  MoveL 8252 to (508.91, 501.9, 16.3) mm, rotated rx 0 ry 90 rz 0 deg; joints [-12.009, -27.828, 110.474, -16.064, -82.068, 51.258]
  Set speed (15.0 mm/s)
  Call Extruder(0.081)
  MoveL 8253 to (508.91, 504.67, 16.3) mm, rotated rx 0 ry 90 rz 0 deg; joints [-12.259, -27.816, 110.402, -16.319, -82.019, 51.306]
  Call Extruder(0.035)
  MoveL 8254 to (507.71, 504.67, 16.3) mm, rotated rx 0 ry 90 rz 0 deg; joints [-12.282, -27.84, 110.547, -16.337, -82.135, 51.275]
  Call Extruder(0.081)
  MoveL 8255 to (507.71, 501.9, 16.3) mm, rotated rx 0 ry 90 rz 0 deg; joints [-12.032, -27.852, 110.619, -16.082, -82.184, 51.227]
  Call Extruder(0.035)
  MoveL 8256 to (508.91, 501.9, 16.3) mm, rotated rx 0 ry 90 rz 0 deg; joints [-12.009, -27.828, 110.474, -16.064, -82.068, 51.258]
  Set speed (120.0 mm/s)
  MoveL 8257 to (508.59, 502.65, 16.3) mm, rotated rx 0 ry 90 rz 0 deg; joints [-12.083, -27.831, 110.493, -16.138, -82.085, 51.263]
  Set speed (15.0 mm/s)
  Call Extruder(0.018)
  MoveL 8258 to (508.15, 502.21, 16.3) mm, rotated rx 0 ry 90 rz 0 deg; joints [-12.052, -27.842, 110.557, -16.105, -82.136, 51.244]
  Set speed (120.0 mm/s)
  MoveL 8259 to (508.02, 503.08, 16.3) mm, rotated rx 0 ry 90 rz 0 deg; joints [-12.132, -27.841, 110.55, -16.186, -82.133, 51.255]
  Set speed (15.0 mm/s)
  Call Extruder(0.023)
  MoveL 8260 to (508.59, 503.64, 16.3) mm, rotated rx 0 ry 90 rz 0 deg; joints [-12.172, -27.827, 110.467, -16.229, -82.068, 51.28]
  Set speed (120.0 mm/s)
  MoveL 8261 to (508.02, 504.07, 16.3) mm, rotated rx 0 ry 90 rz 0 deg; joints [-12.222, -27.836, 110.525, -16.277, -82.116, 51.272]
  Set speed (15.0 mm/s)
  Call Extruder(0.012)
  MoveL 8262 to (508.32, 504.36, 16.3) mm, rotated rx 0 ry 90 rz 0 deg; joints [-12.242, -27.829, 110.482, -16.299, -82.082, 51.285]
  Set speed (120.0 mm/s)
  MoveL 8263 to (490.68, 490.68, 16.3) mm, rotated rx 0 ry 90 rz 0 deg; joints [-11.324, -28.211, 112.929, -15.306, -84.042, 50.621]
  Set speed (1000.0 mm/s)
  MoveL 8264 to (490.68, 490.68, 16.4) mm, rotated rx 0 ry 90 rz 0 deg; joints [-11.324, -28.222, 112.934, -15.306, -84.036, 50.622]
  Set speed (30.0 mm/s)
  Call Extruder(0.767)
  MoveL 8265 to (509.32, 509.32, 16.4) mm, rotated rx 0 ry 90 rz 0 deg; joints [-12.669, -27.797, 110.234, -16.738, -81.892, 51.4]
  MoveL 8266 to (509.44, 509.44, 16.4) mm, rotated rx 0 ry 90 rz 0 deg; joints [-12.677, -27.794, 110.216, -16.747, -81.878, 51.406]
  Set speed (120.0 mm/s)
  MoveL 8267 to (507.79, 502.11, 16.4) mm, rotated rx 0 ry 90 rz 0 deg; joints [-12.049, -27.86, 110.609, -16.101, -82.168, 51.234]
  Set speed (30.0 mm/s)
  Call Extruder(0.297)
  MoveL 8268 to (500.58, 509.32, 16.4) mm, rotated rx 0 ry 90 rz 0 deg; joints [-12.847, -27.971, 111.282, -16.884, -82.735, 51.167]
  Set speed (120.0 mm/s)
  MoveL 8269 to (499.42, 509.32, 16.4) mm, rotated rx 0 ry 90 rz 0 deg; joints [-12.872, -27.993, 111.421, -16.904, -82.847, 51.135]
  Set speed (30.0 mm/s)
  Call Extruder(0.360)
  MoveL 8270 to (490.68, 500.58, 16.4) mm, rotated rx 0 ry 90 rz 0 deg; joints [-12.247, -28.186, 112.689, -16.24, -83.859, 50.763]
  Set speed (120.0 mm/s)
  MoveL 8271 to (490.68, 499.42, 16.4) mm, rotated rx 0 ry 90 rz 0 deg; joints [-12.139, -28.191, 112.719, -16.13, -83.88, 50.746]
  Set speed (30.0 mm/s)
  MoveL 8272 to (499.42, 490.68, 16.4) mm, rotated rx 0 ry 90 rz 0 deg; joints [-11.163, -28.067, 111.894, -15.17, -83.178, 50.841]
  Set speed (120.0 mm/s)
  MoveL 8273 to (500.58, 490.68, 16.4) mm, rotated rx 0 ry 90 rz 0 deg; joints [-11.142, -28.046, 111.756, -15.152, -83.065, 50.869]
  Set speed (30.0 mm/s)
  Call Extruder(0.055)
  MoveL 8274 to (501.92, 492.02, 16.4) mm, rotated rx 0 ry 90 rz 0 deg; joints [-11.24, -28.016, 111.564, -15.257, -82.912, 50.923]
  Set speed (120.0 mm/s)
  MoveL 8275 to (502.08, 492.18, 16.4) mm, rotated rx 0 ry 90 rz 0 deg; joints [-11.252, -28.012, 111.54, -15.27, -82.893, 50.929]
  Set speed (30.0 mm/s)
  Call Extruder(0.298)
  MoveL 8276 to (509.32, 499.42, 16.4) mm, rotated rx 0 ry 90 rz 0 deg; joints [-11.777, -27.841, 110.493, -15.83, -82.065, 51.227]
  Set speed (120.0 mm/s)
  MoveL 8277 to (509.32, 500.58, 16.4) mm, rotated rx 0 ry 90 rz 0 deg; joints [-11.882, -27.836, 110.463, -15.936, -82.046, 51.247]
  Set speed (30.0 mm/s)
  Call Extruder(0.060)
  MoveL 8278 to (507.86, 502.04, 16.4) mm, rotated rx 0 ry 90 rz 0 deg; joints [-12.041, -27.859, 110.602, -16.093, -82.162, 51.235]
  MoveL 8279 to (507.74, 502.16, 16.4) mm, rotated rx 0 ry 90 rz 0 deg; joints [-12.055, -27.861, 110.613, -16.106, -82.172, 51.234]
  Set speed (120.0 mm/s)
  MoveL 8280 to (509.32, 490.68, 16.4) mm, rotated rx 0 ry 90 rz 0 deg; joints [-10.985, -27.876, 110.705, -15.024, -82.209, 51.083]
  Set speed (30.0 mm/s)
  Call Extruder(0.767)
  MoveL 8281 to (490.68, 509.32, 16.4) mm, rotated rx 0 ry 90 rz 0 deg; joints [-13.056, -28.152, 112.457, -17.059, -83.692, 50.896]
  MoveL 8282 to (490.56, 509.44, 16.4) mm, rotated rx 0 ry 90 rz 0 deg; joints [-13.07, -28.154, 112.469, -17.073, -83.701, 50.895]
  Set speed (120.0 mm/s)
  MoveL 8283 to (490.4, 509.6, 16.4) mm, rotated rx 0 ry 90 rz 0 deg; joints [-13.088, -28.156, 112.483, -17.091, -83.713, 50.893]
  Set speed (15.0 mm/s)
  Call Extruder(0.559)
  MoveL 8284 to (490.4, 490.4, 16.4) mm, rotated rx 0 ry 90 rz 0 deg; joints [-11.303, -28.227, 112.973, -15.284, -84.068, 50.611]
  MoveL 8285 to (509.6, 490.4, 16.4) mm, rotated rx 0 ry 90 rz 0 deg; joints [-10.955, -27.872, 110.678, -14.995, -82.186, 51.085]
  MoveL 8286 to (509.6, 509.6, 16.4) mm, rotated rx 0 ry 90 rz 0 deg; joints [-12.688, -27.79, 110.193, -16.759, -81.86, 51.413]
  MoveL 8287 to (490.4, 509.6, 16.4) mm, rotated rx 0 ry 90 rz 0 deg; joints [-13.088, -28.156, 112.483, -17.091, -83.713, 50.893]
  Set speed (120.0 mm/s)
  MoveL 8288 to (490.4, 509.2, 16.4) mm, rotated rx 0 ry 90 rz 0 deg; joints [-13.051, -28.158, 112.494, -17.053, -83.721, 50.887]
  Set speed (1000.0 mm/s)
  MoveL 8289 to (490.5, 509.2, 16.4) mm, rotated rx 0 ry 90 rz 0 deg; joints [-13.049, -28.156, 112.482, -17.052, -83.711, 50.89]
  Set speed (1000.0 mm/s)
  MoveL 8290 to (494.92, 492.25, 16.4) mm, rotated rx 0 ry 90 rz 0 deg; joints [-11.391, -28.143, 112.393, -15.387, -83.593, 50.751]
  Set speed (15.0 mm/s)
  Call Extruder(0.034)
  MoveL 8291 to (494.92, 491.09, 16.4) mm, rotated rx 0 ry 90 rz 0 deg; joints [-11.283, -28.147, 112.421, -15.278, -83.613, 50.735]
  Call Extruder(0.076)
  MoveL 8292 to (497.51, 491.09, 16.4) mm, rotated rx 0 ry 90 rz 0 deg; joints [-11.235, -28.101, 112.112, -15.237, -83.358, 50.799]
  Call Extruder(0.034)
  MoveL 8293 to (497.51, 492.26, 16.4) mm, rotated rx 0 ry 90 rz 0 deg; joints [-11.344, -28.096, 112.084, -15.347, -83.339, 50.817]
  Call Extruder(0.074)
  MoveL 8294 to (494.97, 492.26, 16.4) mm, rotated rx 0 ry 90 rz 0 deg; joints [-11.391, -28.142, 112.387, -15.387, -83.587, 50.753]
  Call Extruder(0.000)
  MoveL 8295 to (494.97, 492.25, 16.4) mm, rotated rx 0 ry 90 rz 0 deg; joints [-11.39, -28.142, 112.387, -15.386, -83.587, 50.753]
  Call Extruder(0.002)
  MoveL 8296 to (494.92, 492.25, 16.4) mm, rotated rx 0 ry 90 rz 0 deg; joints [-11.391, -28.143, 112.393, -15.387, -83.593, 50.751]
  Set speed (120.0 mm/s)
  MoveL 8297 to (495.23, 491.75, 16.4) mm, rotated rx 0 ry 90 rz 0 deg; joints [-11.339, -28.139, 112.368, -15.335, -83.571, 50.752]
  Set speed (15.0 mm/s)
  Call Extruder(0.014)
  MoveL 8298 to (495.58, 491.4, 16.4) mm, rotated rx 0 ry 90 rz 0 deg; joints [-11.3, -28.134, 112.335, -15.297, -83.543, 50.756]
  Set speed (120.0 mm/s)
  MoveL 8299 to (496.02, 491.95, 16.4) mm, rotated rx 0 ry 90 rz 0 deg; joints [-11.342, -28.124, 112.269, -15.341, -83.49, 50.775]
  Set speed (15.0 mm/s)
  Call Extruder(0.022)
  MoveL 8300 to (496.57, 491.4, 16.4) mm, rotated rx 0 ry 90 rz 0 deg; joints [-11.282, -28.117, 112.218, -15.281, -83.446, 50.78]
  Set speed (120.0 mm/s)
  MoveL 8301 to (497.01, 491.95, 16.4) mm, rotated rx 0 ry 90 rz 0 deg; joints [-11.324, -28.107, 112.151, -15.325, -83.393, 50.799]
  Set speed (15.0 mm/s)
  Call Extruder(0.008)
  MoveL 8302 to (497.2, 491.76, 16.4) mm, rotated rx 0 ry 90 rz 0 deg; joints [-11.303, -28.104, 112.134, -15.305, -83.378, 50.801]
  Set speed (120.0 mm/s)
  MoveL 8303 to (501.84, 492.26, 16.4) mm, rotated rx 0 ry 90 rz 0 deg; joints [-11.264, -28.016, 111.568, -15.281, -82.915, 50.924]
  Set speed (15.0 mm/s)
  Call Extruder(0.034)
  MoveL 8304 to (501.84, 491.09, 16.4) mm, rotated rx 0 ry 90 rz 0 deg; joints [-11.157, -28.021, 111.595, -15.172, -82.935, 50.906]
  Call Extruder(0.076)
  MoveL 8305 to (504.46, 491.09, 16.4) mm, rotated rx 0 ry 90 rz 0 deg; joints [-11.109, -27.971, 111.281, -15.133, -82.678, 50.971]
  Call Extruder(0.034)
  MoveL 8306 to (504.46, 492.27, 16.4) mm, rotated rx 0 ry 90 rz 0 deg; joints [-11.217, -27.966, 111.253, -15.242, -82.659, 50.989]
  Call Extruder(0.016)
  MoveL 8307 to (503.92, 492.26, 16.4) mm, rotated rx 0 ry 90 rz 0 deg; joints [-11.226, -27.976, 111.317, -15.25, -82.711, 50.976]
  Call Extruder(0.061)
  MoveL 8308 to (501.84, 492.26, 16.4) mm, rotated rx 0 ry 90 rz 0 deg; joints [-11.264, -28.016, 111.568, -15.281, -82.915, 50.924]
  Set speed (120.0 mm/s)
  MoveL 8309 to (502.15, 491.76, 16.4) mm, rotated rx 0 ry 90 rz 0 deg; joints [-11.212, -28.012, 111.542, -15.229, -82.893, 50.924]
  Set speed (15.0 mm/s)
  Call Extruder(0.015)
  MoveL 8310 to (502.5, 491.4, 16.4) mm, rotated rx 0 ry 90 rz 0 deg; joints [-11.173, -28.007, 111.508, -15.191, -82.864, 50.928]
  Set speed (120.0 mm/s)
  MoveL 8311 to (502.95, 491.95, 16.4) mm, rotated rx 0 ry 90 rz 0 deg; joints [-11.215, -27.996, 111.441, -15.235, -82.811, 50.947]
  Set speed (15.0 mm/s)
  Call Extruder(0.022)
  MoveL 8312 to (503.49, 491.4, 16.4) mm, rotated rx 0 ry 90 rz 0 deg; joints [-11.155, -27.988, 111.389, -15.176, -82.767, 50.952]
  Set speed (120.0 mm/s)
  MoveL 8313 to (503.94, 491.95, 16.4) mm, rotated rx 0 ry 90 rz 0 deg; joints [-11.197, -27.977, 111.323, -15.22, -82.714, 50.972]
  Set speed (15.0 mm/s)
  Call Extruder(0.008)
  MoveL 8314 to (504.14, 491.75, 16.4) mm, rotated rx 0 ry 90 rz 0 deg; joints [-11.175, -27.974, 111.303, -15.198, -82.698, 50.973]
  Set speed (120.0 mm/s)
  MoveL 8315 to (507.71, 494.38, 16.4) mm, rotated rx 0 ry 90 rz 0 deg; joints [-11.351, -27.894, 110.81, -15.39, -82.306, 51.104]
  Set speed (15.0 mm/s)
  Call Extruder(0.035)
  MoveL 8316 to (508.91, 494.38, 16.4) mm, rotated rx 0 ry 90 rz 0 deg; joints [-11.328, -27.87, 110.667, -15.371, -82.189, 51.133]
  Call Extruder(0.079)
  MoveL 8317 to (508.91, 497.08, 16.4) mm, rotated rx 0 ry 90 rz 0 deg; joints [-11.573, -27.859, 110.601, -15.62, -82.145, 51.178]
  Call Extruder(0.035)
  MoveL 8318 to (507.71, 497.08, 16.4) mm, rotated rx 0 ry 90 rz 0 deg; joints [-11.595, -27.883, 110.745, -15.638, -82.261, 51.148]
  Call Extruder(0.051)
  MoveL 8319 to (507.71, 495.33, 16.4) mm, rotated rx 0 ry 90 rz 0 deg; joints [-11.437, -27.89, 110.788, -15.477, -82.29, 51.119]
  Call Extruder(0.028)
  MoveL 8320 to (507.71, 494.38, 16.4) mm, rotated rx 0 ry 90 rz 0 deg; joints [-11.351, -27.894, 110.81, -15.39, -82.306, 51.104]
  Set speed (120.0 mm/s)
  MoveL 8321 to (508.59, 495.21, 16.4) mm, rotated rx 0 ry 90 rz 0 deg; joints [-11.41, -27.873, 110.684, -15.453, -82.206, 51.139]
  Set speed (15.0 mm/s)
  Call Extruder(0.023)
  MoveL 8322 to (508.03, 495.78, 16.4) mm, rotated rx 0 ry 90 rz 0 deg; joints [-11.472, -27.882, 110.739, -15.514, -82.252, 51.134]
  Set speed (120.0 mm/s)
  MoveL 8323 to (508.59, 496.2, 16.4) mm, rotated rx 0 ry 90 rz 0 deg; joints [-11.5, -27.869, 110.66, -15.545, -82.19, 51.155]
  Set speed (15.0 mm/s)
  Call Extruder(0.023)
  MoveL 8324 to (508.04, 496.76, 16.4) mm, rotated rx 0 ry 90 rz 0 deg; joints [-11.56, -27.878, 110.714, -15.604, -82.235, 51.151]
  Set speed (120.0 mm/s)
  MoveL 8325 to (507.71, 501.95, 16.4) mm, rotated rx 0 ry 90 rz 0 deg; joints [-12.037, -27.862, 110.622, -16.088, -82.178, 51.23]
  Set speed (15.0 mm/s)
  Call Extruder(0.035)
  MoveL 8326 to (508.91, 501.96, 16.4) mm, rotated rx 0 ry 90 rz 0 deg; joints [-12.014, -27.838, 110.478, -16.069, -82.062, 51.26]
  Call Extruder(0.079)
  MoveL 8327 to (508.91, 504.67, 16.4) mm, rotated rx 0 ry 90 rz 0 deg; joints [-12.259, -27.826, 110.407, -16.319, -82.014, 51.307]
  Call Extruder(0.035)
  MoveL 8328 to (507.71, 504.67, 16.4) mm, rotated rx 0 ry 90 rz 0 deg; joints [-12.282, -27.851, 110.552, -16.338, -82.13, 51.276]
  Call Extruder(0.079)
  MoveL 8329 to (507.71, 501.95, 16.4) mm, rotated rx 0 ry 90 rz 0 deg; joints [-12.037, -27.862, 110.622, -16.088, -82.178, 51.23]
  Set speed (120.0 mm/s)
  MoveL 8330 to (508.03, 502.71, 16.4) mm, rotated rx 0 ry 90 rz 0 deg; joints [-12.099, -27.853, 110.565, -16.153, -82.134, 51.251]
  Set speed (15.0 mm/s)
  Call Extruder(0.018)
  MoveL 8331 to (508.47, 502.27, 16.4) mm, rotated rx 0 ry 90 rz 0 deg; joints [-12.051, -27.846, 110.523, -16.105, -82.099, 51.254]
  Set speed (120.0 mm/s)
  MoveL 8332 to (508.59, 503.13, 16.4) mm, rotated rx 0 ry 90 rz 0 deg; joints [-12.126, -27.839, 110.485, -16.182, -82.072, 51.273]
  Set speed (15.0 mm/s)
  Call Extruder(0.023)
  MoveL 8333 to (508.02, 503.7, 16.4) mm, rotated rx 0 ry 90 rz 0 deg; joints [-12.189, -27.848, 110.539, -16.244, -82.117, 51.268]
  Set speed (120.0 mm/s)
  MoveL 8334 to (508.59, 504.12, 16.4) mm, rotated rx 0 ry 90 rz 0 deg; joints [-12.216, -27.835, 110.46, -16.273, -82.054, 51.29]
  Set speed (15.0 mm/s)
  Call Extruder(0.010)
  MoveL 8335 to (508.36, 504.36, 16.4) mm, rotated rx 0 ry 90 rz 0 deg; joints [-12.241, -27.839, 110.482, -16.299, -82.073, 51.288]
  Set speed (120.0 mm/s)
  MoveL 8336 to (490.68, 490.68, 16.4) mm, rotated rx 0 ry 90 rz 0 deg; joints [-11.324, -28.222, 112.934, -15.306, -84.036, 50.622]
  Set speed (1000.0 mm/s)
  MoveL 8337 to (490.68, 490.68, 16.5) mm, rotated rx 0 ry 90 rz 0 deg; joints [-11.324, -28.232, 112.939, -15.306, -84.031, 50.624]
  Set speed (30.0 mm/s)
  Call Extruder(0.767)
  MoveL 8338 to (509.32, 509.32, 16.5) mm, rotated rx 0 ry 90 rz 0 deg; joints [-12.669, -27.807, 110.239, -16.738, -81.887, 51.402]
  MoveL 8339 to (509.44, 509.44, 16.5) mm, rotated rx 0 ry 90 rz 0 deg; joints [-12.677, -27.804, 110.221, -16.747, -81.873, 51.407]
  Set speed (120.0 mm/s)
  MoveL 8340 to (507.79, 502.11, 16.5) mm, rotated rx 0 ry 90 rz 0 deg; joints [-12.049, -27.871, 110.614, -16.101, -82.162, 51.236]
  Set speed (30.0 mm/s)
  Call Extruder(0.297)
  MoveL 8341 to (500.58, 509.32, 16.5) mm, rotated rx 0 ry 90 rz 0 deg; joints [-12.847, -27.981, 111.287, -16.884, -82.73, 51.168]
  Set speed (120.0 mm/s)
  MoveL 8342 to (499.42, 509.32, 16.5) mm, rotated rx 0 ry 90 rz 0 deg; joints [-12.872, -28.003, 111.426, -16.904, -82.842, 51.137]
  Set speed (30.0 mm/s)
  Call Extruder(0.360)
  MoveL 8343 to (490.68, 500.58, 16.5) mm, rotated rx 0 ry 90 rz 0 deg; joints [-12.247, -28.197, 112.694, -16.24, -83.853, 50.765]
  Set speed (120.0 mm/s)
  MoveL 8344 to (490.68, 499.42, 16.5) mm, rotated rx 0 ry 90 rz 0 deg; joints [-12.139, -28.201, 112.724, -16.131, -83.875, 50.748]
  Set speed (30.0 mm/s)
  MoveL 8345 to (499.42, 490.68, 16.5) mm, rotated rx 0 ry 90 rz 0 deg; joints [-11.163, -28.078, 111.899, -15.17, -83.173, 50.842]
  Set speed (120.0 mm/s)
  MoveL 8346 to (500.58, 490.68, 16.5) mm, rotated rx 0 ry 90 rz 0 deg; joints [-11.141, -28.056, 111.761, -15.152, -83.059, 50.871]
  Set speed (30.0 mm/s)
  Call Extruder(0.058)
  MoveL 8347 to (501.98, 492.08, 16.5) mm, rotated rx 0 ry 90 rz 0 deg; joints [-11.245, -28.025, 111.56, -15.262, -82.899, 50.927]
  Set speed (120.0 mm/s)
  MoveL 8348 to (502.08, 492.18, 16.5) mm, rotated rx 0 ry 90 rz 0 deg; joints [-11.252, -28.022, 111.545, -15.27, -82.887, 50.931]
  Set speed (30.0 mm/s)
  Call Extruder(0.298)
  MoveL 8349 to (509.32, 499.42, 16.5) mm, rotated rx 0 ry 90 rz 0 deg; joints [-11.777, -27.851, 110.498, -15.83, -82.06, 51.229]
  Set speed (120.0 mm/s)
  MoveL 8350 to (509.32, 500.58, 16.5) mm, rotated rx 0 ry 90 rz 0 deg; joints [-11.882, -27.846, 110.469, -15.937, -82.04, 51.249]
  Set speed (30.0 mm/s)
  Call Extruder(0.062)
  MoveL 8351 to (507.81, 502.09, 16.5) mm, rotated rx 0 ry 90 rz 0 deg; joints [-12.047, -27.87, 110.612, -16.099, -82.161, 51.236]
  MoveL 8352 to (507.69, 502.21, 16.5) mm, rotated rx 0 ry 90 rz 0 deg; joints [-12.061, -27.872, 110.624, -16.112, -82.171, 51.235]
  Set speed (120.0 mm/s)
  MoveL 8353 to (509.32, 490.68, 16.5) mm, rotated rx 0 ry 90 rz 0 deg; joints [-10.985, -27.887, 110.71, -15.025, -82.204, 51.084]
  Set speed (30.0 mm/s)
  Call Extruder(0.767)
  MoveL 8354 to (490.68, 509.32, 16.5) mm, rotated rx 0 ry 90 rz 0 deg; joints [-13.056, -28.163, 112.463, -17.06, -83.686, 50.898]
  MoveL 8355 to (490.56, 509.44, 16.5) mm, rotated rx 0 ry 90 rz 0 deg; joints [-13.07, -28.165, 112.474, -17.073, -83.696, 50.897]
  Set speed (120.0 mm/s)
  MoveL 8356 to (490.4, 509.6, 16.5) mm, rotated rx 0 ry 90 rz 0 deg; joints [-13.088, -28.167, 112.488, -17.091, -83.708, 50.895]
  Set speed (15.0 mm/s)
  Call Extruder(0.559)
  MoveL 8357 to (490.4, 490.4, 16.5) mm, rotated rx 0 ry 90 rz 0 deg; joints [-11.303, -28.238, 112.978, -15.284, -84.063, 50.613]
  MoveL 8358 to (509.6, 490.4, 16.5) mm, rotated rx 0 ry 90 rz 0 deg; joints [-10.955, -27.882, 110.683, -14.995, -82.181, 51.086]
  MoveL 8359 to (509.6, 509.6, 16.5) mm, rotated rx 0 ry 90 rz 0 deg; joints [-12.688, -27.8, 110.198, -16.759, -81.855, 51.414]
  MoveL 8360 to (490.4, 509.6, 16.5) mm, rotated rx 0 ry 90 rz 0 deg; joints [-13.088, -28.167, 112.488, -17.091, -83.708, 50.895]
  Set speed (120.0 mm/s)
  MoveL 8361 to (490.4, 509.2, 16.5) mm, rotated rx 0 ry 90 rz 0 deg; joints [-13.051, -28.168, 112.499, -17.054, -83.716, 50.888]
  Set speed (1000.0 mm/s)
  MoveL 8362 to (490.5, 509.2, 16.5) mm, rotated rx 0 ry 90 rz 0 deg; joints [-13.049, -28.167, 112.487, -17.052, -83.706, 50.891]
  Set speed (1000.0 mm/s)
  MoveL 8363 to (494.92, 492.25, 16.5) mm, rotated rx 0 ry 90 rz 0 deg; joints [-11.391, -28.154, 112.399, -15.387, -83.588, 50.753]
  Set speed (15.0 mm/s)
  Call Extruder(0.034)
  MoveL 8364 to (494.92, 491.09, 16.5) mm, rotated rx 0 ry 90 rz 0 deg; joints [-11.283, -28.158, 112.426, -15.278, -83.608, 50.736]
  Call Extruder(0.074)
  MoveL 8365 to (497.46, 491.09, 16.5) mm, rotated rx 0 ry 90 rz 0 deg; joints [-11.236, -28.112, 112.124, -15.238, -83.358, 50.799]
  Call Extruder(0.034)
  MoveL 8366 to (497.45, 492.26, 16.5) mm, rotated rx 0 ry 90 rz 0 deg; joints [-11.345, -28.108, 112.096, -15.348, -83.339, 50.817]
  Call Extruder(0.072)
  MoveL 8367 to (494.97, 492.26, 16.5) mm, rotated rx 0 ry 90 rz 0 deg; joints [-11.391, -28.152, 112.392, -15.387, -83.582, 50.754]
  Call Extruder(0.000)
  MoveL 8368 to (494.97, 492.25, 16.5) mm, rotated rx 0 ry 90 rz 0 deg; joints [-11.39, -28.153, 112.392, -15.386, -83.582, 50.754]
  Call Extruder(0.002)
  MoveL 8369 to (494.92, 492.25, 16.5) mm, rotated rx 0 ry 90 rz 0 deg; joints [-11.391, -28.154, 112.399, -15.387, -83.588, 50.753]
  Set speed (120.0 mm/s)
  MoveL 8370 to (495.37, 491.41, 16.5) mm, rotated rx 0 ry 90 rz 0 deg; joints [-11.304, -28.149, 112.365, -15.3, -83.558, 50.752]
  Set speed (15.0 mm/s)
  Call Extruder(0.022)
  MoveL 8371 to (495.91, 491.95, 16.5) mm, rotated rx 0 ry 90 rz 0 deg; joints [-11.344, -28.137, 112.288, -15.343, -83.496, 50.773]
  Set speed (120.0 mm/s)
  MoveL 8372 to (496.36, 491.41, 16.5) mm, rotated rx 0 ry 90 rz 0 deg; joints [-11.286, -28.131, 112.248, -15.285, -83.461, 50.777]
  Set speed (15.0 mm/s)
  MoveL 8373 to (496.9, 491.95, 16.5) mm, rotated rx 0 ry 90 rz 0 deg; joints [-11.326, -28.119, 112.17, -15.327, -83.399, 50.798]
  Set speed (120.0 mm/s)
  MoveL 8374 to (501.9, 492.26, 16.5) mm, rotated rx 0 ry 90 rz 0 deg; joints [-11.263, -28.026, 111.565, -15.28, -82.904, 50.927]
  Set speed (15.0 mm/s)
  Call Extruder(0.034)
  MoveL 8375 to (501.9, 491.09, 16.5) mm, rotated rx 0 ry 90 rz 0 deg; joints [-11.155, -28.03, 111.593, -15.171, -82.923, 50.909]
  Call Extruder(0.074)
  MoveL 8376 to (504.46, 491.09, 16.5) mm, rotated rx 0 ry 90 rz 0 deg; joints [-11.109, -27.981, 111.286, -15.133, -82.673, 50.972]
  Call Extruder(0.034)
  MoveL 8377 to (504.46, 492.27, 16.5) mm, rotated rx 0 ry 90 rz 0 deg; joints [-11.217, -27.977, 111.258, -15.243, -82.653, 50.991]
  Call Extruder(0.016)
  MoveL 8378 to (503.92, 492.26, 16.5) mm, rotated rx 0 ry 90 rz 0 deg; joints [-11.226, -27.987, 111.323, -15.25, -82.706, 50.977]
  Call Extruder(0.059)
  MoveL 8379 to (501.9, 492.26, 16.5) mm, rotated rx 0 ry 90 rz 0 deg; joints [-11.263, -28.026, 111.565, -15.28, -82.904, 50.927]
  Set speed (120.0 mm/s)
  MoveL 8380 to (502.29, 491.4, 16.5) mm, rotated rx 0 ry 90 rz 0 deg; joints [-11.177, -28.021, 111.538, -15.194, -82.879, 50.924]
  Set speed (15.0 mm/s)
  Call Extruder(0.022)
  MoveL 8381 to (502.84, 491.95, 16.5) mm, rotated rx 0 ry 90 rz 0 deg; joints [-11.217, -28.009, 111.46, -15.237, -82.817, 50.946]
  Set speed (120.0 mm/s)
  MoveL 8382 to (503.28, 491.4, 16.5) mm, rotated rx 0 ry 90 rz 0 deg; joints [-11.159, -28.002, 111.42, -15.18, -82.782, 50.948]
  Set speed (15.0 mm/s)
  Call Extruder(0.022)
  MoveL 8383 to (503.82, 491.95, 16.5) mm, rotated rx 0 ry 90 rz 0 deg; joints [-11.199, -27.99, 111.342, -15.222, -82.721, 50.97]
  Set speed (120.0 mm/s)
  MoveL 8384 to (507.72, 494.39, 16.5) mm, rotated rx 0 ry 90 rz 0 deg; joints [-11.351, -27.904, 110.815, -15.39, -82.3, 51.105]
  Set speed (15.0 mm/s)
  Call Extruder(0.035)
  MoveL 8385 to (508.91, 494.38, 16.5) mm, rotated rx 0 ry 90 rz 0 deg; joints [-11.328, -27.88, 110.672, -15.372, -82.184, 51.134]
  Call Extruder(0.077)
  MoveL 8386 to (508.91, 497.02, 16.5) mm, rotated rx 0 ry 90 rz 0 deg; joints [-11.568, -27.869, 110.607, -15.615, -82.14, 51.178]
  Call Extruder(0.035)
  MoveL 8387 to (507.71, 497.02, 16.5) mm, rotated rx 0 ry 90 rz 0 deg; joints [-11.59, -27.894, 110.751, -15.633, -82.257, 51.148]
  Call Extruder(0.077)
  MoveL 8388 to (507.72, 494.39, 16.5) mm, rotated rx 0 ry 90 rz 0 deg; joints [-11.351, -27.904, 110.815, -15.39, -82.3, 51.105]
  Set speed (120.0 mm/s)
  MoveL 8389 to (508.03, 495.16, 16.5) mm, rotated rx 0 ry 90 rz 0 deg; joints [-11.415, -27.895, 110.759, -15.457, -82.257, 51.125]
  Set speed (15.0 mm/s)
  Call Extruder(0.023)
  MoveL 8390 to (508.59, 495.72, 16.5) mm, rotated rx 0 ry 90 rz 0 deg; joints [-11.456, -27.881, 110.677, -15.501, -82.193, 51.149]
  Set speed (120.0 mm/s)
  MoveL 8391 to (508.03, 496.15, 16.5) mm, rotated rx 0 ry 90 rz 0 deg; joints [-11.505, -27.891, 110.735, -15.548, -82.241, 51.142]
  Set speed (15.0 mm/s)
  Call Extruder(0.023)
  MoveL 8392 to (508.58, 496.7, 16.5) mm, rotated rx 0 ry 90 rz 0 deg; joints [-11.545, -27.877, 110.654, -15.591, -82.178, 51.165]
  Set speed (120.0 mm/s)
  MoveL 8393 to (508.91, 502.01, 16.5) mm, rotated rx 0 ry 90 rz 0 deg; joints [-12.019, -27.848, 110.481, -16.075, -82.056, 51.263]
  Set speed (15.0 mm/s)
  Call Extruder(0.077)
  MoveL 8394 to (508.91, 504.67, 16.5) mm, rotated rx 0 ry 90 rz 0 deg; joints [-12.259, -27.837, 110.412, -16.319, -82.009, 51.309]
  Call Extruder(0.035)
  MoveL 8395 to (507.71, 504.67, 16.5) mm, rotated rx 0 ry 90 rz 0 deg; joints [-12.282, -27.861, 110.557, -16.338, -82.125, 51.278]
  Call Extruder(0.077)
  MoveL 8396 to (507.71, 502.01, 16.5) mm, rotated rx 0 ry 90 rz 0 deg; joints [-12.042, -27.873, 110.626, -16.093, -82.172, 51.232]
  Call Extruder(0.035)
  MoveL 8397 to (508.91, 502.01, 16.5) mm, rotated rx 0 ry 90 rz 0 deg; joints [-12.019, -27.848, 110.481, -16.075, -82.056, 51.263]
  Set speed (120.0 mm/s)
  MoveL 8398 to (508.59, 502.65, 16.5) mm, rotated rx 0 ry 90 rz 0 deg; joints [-12.083, -27.852, 110.503, -16.139, -82.075, 51.266]
  Set speed (15.0 mm/s)
  Call Extruder(0.014)
  MoveL 8399 to (508.26, 502.33, 16.5) mm, rotated rx 0 ry 90 rz 0 deg; joints [-12.06, -27.86, 110.551, -16.113, -82.113, 51.252]
  Set speed (120.0 mm/s)
  MoveL 8400 to (508.02, 503.08, 16.5) mm, rotated rx 0 ry 90 rz 0 deg; joints [-12.132, -27.862, 110.561, -16.186, -82.123, 51.258]
  Set speed (15.0 mm/s)
  Call Extruder(0.023)
  MoveL 8401 to (508.59, 503.64, 16.5) mm, rotated rx 0 ry 90 rz 0 deg; joints [-12.172, -27.848, 110.477, -16.229, -82.058, 51.283]
  Set speed (120.0 mm/s)
  MoveL 8402 to (508.03, 504.07, 16.5) mm, rotated rx 0 ry 90 rz 0 deg; joints [-12.222, -27.857, 110.535, -16.277, -82.105, 51.275]
  Set speed (15.0 mm/s)
  Call Extruder(0.012)
  MoveL 8403 to (508.32, 504.36, 16.5) mm, rotated rx 0 ry 90 rz 0 deg; joints [-12.242, -27.85, 110.492, -16.299, -82.072, 51.288]
  Set speed (120.0 mm/s)
  MoveL 8404 to (490.68, 490.68, 16.5) mm, rotated rx 0 ry 90 rz 0 deg; joints [-11.324, -28.232, 112.939, -15.306, -84.031, 50.624]
  Set speed (1000.0 mm/s)
  MoveL 8405 to (490.68, 490.68, 16.6) mm, rotated rx 0 ry 90 rz 0 deg; joints [-11.324, -28.243, 112.944, -15.306, -84.026, 50.625]
  Set speed (30.0 mm/s)
  Call Extruder(0.767)
  MoveL 8406 to (509.32, 509.32, 16.6) mm, rotated rx 0 ry 90 rz 0 deg; joints [-12.669, -27.818, 110.244, -16.738, -81.882, 51.404]
  MoveL 8407 to (509.44, 509.44, 16.6) mm, rotated rx 0 ry 90 rz 0 deg; joints [-12.677, -27.814, 110.226, -16.748, -81.867, 51.409]
  Set speed (120.0 mm/s)
  MoveL 8408 to (500.58, 509.32, 16.6) mm, rotated rx 0 ry 90 rz 0 deg; joints [-12.847, -27.992, 111.293, -16.884, -82.725, 51.17]
  Set speed (30.0 mm/s)
  Call Extruder(0.360)
  MoveL 8409 to (509.32, 500.58, 16.6) mm, rotated rx 0 ry 90 rz 0 deg; joints [-11.882, -27.857, 110.474, -15.937, -82.035, 51.25]
  Set speed (120.0 mm/s)
  MoveL 8410 to (509.32, 499.42, 16.6) mm, rotated rx 0 ry 90 rz 0 deg; joints [-11.777, -27.862, 110.503, -15.83, -82.055, 51.23]
  Set speed (30.0 mm/s)
  Call Extruder(0.298)
  MoveL 8411 to (502.08, 492.18, 16.6) mm, rotated rx 0 ry 90 rz 0 deg; joints [-11.252, -28.033, 111.55, -15.27, -82.882, 50.932]
  Set speed (120.0 mm/s)
  MoveL 8412 to (502.04, 492.14, 16.6) mm, rotated rx 0 ry 90 rz 0 deg; joints [-11.249, -28.034, 111.556, -15.267, -82.887, 50.931]
  Set speed (30.0 mm/s)
  Call Extruder(0.060)
  MoveL 8413 to (500.58, 490.68, 16.6) mm, rotated rx 0 ry 90 rz 0 deg; joints [-11.142, -28.067, 111.766, -15.153, -83.054, 50.872]
  Set speed (120.0 mm/s)
  MoveL 8414 to (499.42, 490.68, 16.6) mm, rotated rx 0 ry 90 rz 0 deg; joints [-11.163, -28.088, 111.904, -15.17, -83.168, 50.844]
  Set speed (30.0 mm/s)
  Call Extruder(0.360)
  MoveL 8415 to (490.68, 499.42, 16.6) mm, rotated rx 0 ry 90 rz 0 deg; joints [-12.139, -28.212, 112.729, -16.131, -83.869, 50.749]
  Set speed (120.0 mm/s)
  MoveL 8416 to (490.68, 500.58, 16.6) mm, rotated rx 0 ry 90 rz 0 deg; joints [-12.247, -28.208, 112.7, -16.24, -83.848, 50.766]
  Set speed (30.0 mm/s)
  MoveL 8417 to (499.42, 509.32, 16.6) mm, rotated rx 0 ry 90 rz 0 deg; joints [-12.872, -28.014, 111.431, -16.904, -82.836, 51.139]
  MoveL 8418 to (499.54, 509.44, 16.6) mm, rotated rx 0 ry 90 rz 0 deg; joints [-12.88, -28.011, 111.413, -16.914, -82.822, 51.144]
  Set speed (120.0 mm/s)
  MoveL 8419 to (490.68, 509.32, 16.6) mm, rotated rx 0 ry 90 rz 0 deg; joints [-13.056, -28.174, 112.468, -17.06, -83.681, 50.9]
  Set speed (30.0 mm/s)
  Call Extruder(0.767)
  MoveL 8420 to (509.32, 490.68, 16.6) mm, rotated rx 0 ry 90 rz 0 deg; joints [-10.985, -27.897, 110.715, -15.025, -82.199, 51.085]
  MoveL 8421 to (509.44, 490.56, 16.6) mm, rotated rx 0 ry 90 rz 0 deg; joints [-10.972, -27.895, 110.703, -15.012, -82.189, 51.086]
  Set speed (120.0 mm/s)
  MoveL 8422 to (490.47, 509.53, 16.6) mm, rotated rx 0 ry 90 rz 0 deg; joints [-13.08, -28.176, 112.487, -17.083, -83.697, 50.897]
  Set speed (1000.0 mm/s)
  MoveL 8423 to (490.4, 509.6, 16.6) mm, rotated rx 0 ry 90 rz 0 deg; joints [-13.088, -28.177, 112.493, -17.091, -83.703, 50.896]
  Set speed (15.0 mm/s)
  Call Extruder(0.559)
  MoveL 8424 to (490.4, 490.4, 16.6) mm, rotated rx 0 ry 90 rz 0 deg; joints [-11.303, -28.249, 112.984, -15.284, -84.058, 50.614]
  MoveL 8425 to (509.6, 490.4, 16.6) mm, rotated rx 0 ry 90 rz 0 deg; joints [-10.955, -27.893, 110.688, -14.995, -82.176, 51.088]
  MoveL 8426 to (509.6, 509.6, 16.6) mm, rotated rx 0 ry 90 rz 0 deg; joints [-12.688, -27.81, 110.203, -16.759, -81.849, 51.416]
  MoveL 8427 to (490.4, 509.6, 16.6) mm, rotated rx 0 ry 90 rz 0 deg; joints [-13.088, -28.177, 112.493, -17.091, -83.703, 50.896]
  Set speed (120.0 mm/s)
  MoveL 8428 to (490.4, 509.2, 16.6) mm, rotated rx 0 ry 90 rz 0 deg; joints [-13.051, -28.179, 112.504, -17.054, -83.711, 50.89]
  Set speed (1000.0 mm/s)
  MoveL 8429 to (490.5, 509.2, 16.6) mm, rotated rx 0 ry 90 rz 0 deg; joints [-13.049, -28.177, 112.492, -17.052, -83.701, 50.893]
  Set speed (1000.0 mm/s)
  MoveL 8430 to (494.92, 492.25, 16.6) mm, rotated rx 0 ry 90 rz 0 deg; joints [-11.391, -28.164, 112.404, -15.387, -83.582, 50.754]
  Set speed (15.0 mm/s)
  Call Extruder(0.034)
  MoveL 8431 to (494.92, 491.09, 16.6) mm, rotated rx 0 ry 90 rz 0 deg; joints [-11.283, -28.168, 112.431, -15.278, -83.602, 50.738]
  Call Extruder(0.072)
  MoveL 8432 to (497.4, 491.09, 16.6) mm, rotated rx 0 ry 90 rz 0 deg; joints [-11.237, -28.124, 112.136, -15.239, -83.359, 50.8]
  Call Extruder(0.034)
  MoveL 8433 to (497.4, 492.26, 16.6) mm, rotated rx 0 ry 90 rz 0 deg; joints [-11.346, -28.12, 112.108, -15.349, -83.339, 50.817]
  Call Extruder(0.071)
  MoveL 8434 to (494.97, 492.26, 16.6) mm, rotated rx 0 ry 90 rz 0 deg; joints [-11.391, -28.163, 112.397, -15.387, -83.577, 50.756]
  Call Extruder(0.000)
  MoveL 8435 to (494.97, 492.25, 16.6) mm, rotated rx 0 ry 90 rz 0 deg; joints [-11.39, -28.163, 112.397, -15.386, -83.577, 50.756]
  Call Extruder(0.002)
  MoveL 8436 to (494.92, 492.25, 16.6) mm, rotated rx 0 ry 90 rz 0 deg; joints [-11.391, -28.164, 112.404, -15.387, -83.582, 50.754]
  Set speed (120.0 mm/s)
  MoveL 8437 to (495.23, 491.75, 16.6) mm, rotated rx 0 ry 90 rz 0 deg; joints [-11.339, -28.16, 112.378, -15.335, -83.56, 50.755]
  Set speed (15.0 mm/s)
  Call Extruder(0.014)
  MoveL 8438 to (495.58, 491.4, 16.6) mm, rotated rx 0 ry 90 rz 0 deg; joints [-11.3, -28.155, 112.346, -15.297, -83.532, 50.759]
  Set speed (120.0 mm/s)
  MoveL 8439 to (496.02, 491.95, 16.6) mm, rotated rx 0 ry 90 rz 0 deg; joints [-11.342, -28.146, 112.28, -15.341, -83.479, 50.778]
  Set speed (15.0 mm/s)
  Call Extruder(0.022)
  MoveL 8440 to (496.56, 491.4, 16.6) mm, rotated rx 0 ry 90 rz 0 deg; joints [-11.282, -28.138, 112.228, -15.282, -83.435, 50.783]
  Set speed (120.0 mm/s)
  MoveL 8441 to (501.96, 491.09, 16.6) mm, rotated rx 0 ry 90 rz 0 deg; joints [-11.154, -28.039, 111.59, -15.17, -82.912, 50.912]
  Set speed (15.0 mm/s)
  Call Extruder(0.073)
  MoveL 8442 to (504.46, 491.09, 16.6) mm, rotated rx 0 ry 90 rz 0 deg; joints [-11.109, -27.992, 111.291, -15.133, -82.667, 50.974]
  Call Extruder(0.034)
  MoveL 8443 to (504.46, 492.27, 16.6) mm, rotated rx 0 ry 90 rz 0 deg; joints [-11.217, -27.987, 111.263, -15.243, -82.648, 50.992]
  Call Extruder(0.016)
  MoveL 8444 to (503.92, 492.26, 16.6) mm, rotated rx 0 ry 90 rz 0 deg; joints [-11.226, -27.998, 111.328, -15.25, -82.701, 50.979]
  Call Extruder(0.057)
  MoveL 8445 to (501.96, 492.26, 16.6) mm, rotated rx 0 ry 90 rz 0 deg; joints [-11.262, -28.035, 111.563, -15.279, -82.892, 50.93]
  Call Extruder(0.034)
  MoveL 8446 to (501.96, 491.09, 16.6) mm, rotated rx 0 ry 90 rz 0 deg; joints [-11.154, -28.039, 111.59, -15.17, -82.912, 50.912]
  Set speed (120.0 mm/s)
  MoveL 8447 to (502.28, 491.63, 16.6) mm, rotated rx 0 ry 90 rz 0 deg; joints [-11.198, -28.031, 111.54, -15.216, -82.872, 50.929]
  Set speed (15.0 mm/s)
  Call Extruder(0.009)
  MoveL 8448 to (502.5, 491.4, 16.6) mm, rotated rx 0 ry 90 rz 0 deg; joints [-11.173, -28.028, 111.518, -15.191, -82.853, 50.931]
  Set speed (120.0 mm/s)
  MoveL 8449 to (502.95, 491.95, 16.6) mm, rotated rx 0 ry 90 rz 0 deg; joints [-11.215, -28.017, 111.451, -15.235, -82.801, 50.95]
  Set speed (15.0 mm/s)
  Call Extruder(0.022)
  MoveL 8450 to (503.49, 491.4, 16.6) mm, rotated rx 0 ry 90 rz 0 deg; joints [-11.155, -28.009, 111.399, -15.177, -82.757, 50.955]
  Set speed (120.0 mm/s)
  MoveL 8451 to (503.94, 491.95, 16.6) mm, rotated rx 0 ry 90 rz 0 deg; joints [-11.197, -27.998, 111.333, -15.22, -82.704, 50.974]
  Set speed (15.0 mm/s)
  Call Extruder(0.008)
  MoveL 8452 to (504.14, 491.75, 16.6) mm, rotated rx 0 ry 90 rz 0 deg; joints [-11.175, -27.995, 111.313, -15.199, -82.688, 50.976]
  Set speed (120.0 mm/s)
  MoveL 8453 to (507.72, 494.39, 16.6) mm, rotated rx 0 ry 90 rz 0 deg; joints [-11.351, -27.915, 110.82, -15.39, -82.295, 51.107]
  Set speed (15.0 mm/s)
  Call Extruder(0.035)
  MoveL 8454 to (508.91, 494.38, 16.6) mm, rotated rx 0 ry 90 rz 0 deg; joints [-11.328, -27.891, 110.677, -15.372, -82.179, 51.136]
  Call Extruder(0.075)
  MoveL 8455 to (508.91, 496.96, 16.6) mm, rotated rx 0 ry 90 rz 0 deg; joints [-11.562, -27.88, 110.614, -15.61, -82.136, 51.179]
  Call Extruder(0.035)
  MoveL 8456 to (507.71, 496.96, 16.6) mm, rotated rx 0 ry 90 rz 0 deg; joints [-11.584, -27.904, 110.758, -15.628, -82.253, 51.149]
  Call Extruder(0.051)
  MoveL 8457 to (507.72, 495.21, 16.6) mm, rotated rx 0 ry 90 rz 0 deg; joints [-11.426, -27.911, 110.8, -15.467, -82.282, 51.12]
  Call Extruder(0.024)
  MoveL 8458 to (507.72, 494.39, 16.6) mm, rotated rx 0 ry 90 rz 0 deg; joints [-11.351, -27.915, 110.82, -15.39, -82.295, 51.107]
  Set speed (120.0 mm/s)
  MoveL 8459 to (508.59, 495.21, 16.6) mm, rotated rx 0 ry 90 rz 0 deg; joints [-11.41, -27.894, 110.694, -15.454, -82.196, 51.142]
  Set speed (15.0 mm/s)
  Call Extruder(0.023)
  MoveL 8460 to (508.03, 495.78, 16.6) mm, rotated rx 0 ry 90 rz 0 deg; joints [-11.472, -27.903, 110.749, -15.514, -82.242, 51.137]
  Set speed (120.0 mm/s)
  MoveL 8461 to (508.59, 496.2, 16.6) mm, rotated rx 0 ry 90 rz 0 deg; joints [-11.5, -27.89, 110.67, -15.545, -82.179, 51.158]
  Set speed (15.0 mm/s)
  Call Extruder(0.018)
  MoveL 8462 to (508.15, 496.64, 16.6) mm, rotated rx 0 ry 90 rz 0 deg; joints [-11.548, -27.897, 110.712, -15.592, -82.215, 51.155]
  Set speed (120.0 mm/s)
  MoveL 8463 to (507.71, 502.07, 16.6) mm, rotated rx 0 ry 90 rz 0 deg; joints [-12.047, -27.883, 110.629, -16.098, -82.165, 51.235]
  Set speed (15.0 mm/s)
  Call Extruder(0.035)
  MoveL 8464 to (508.91, 502.07, 16.6) mm, rotated rx 0 ry 90 rz 0 deg; joints [-12.024, -27.859, 110.485, -16.08, -82.049, 51.265]
  Call Extruder(0.076)
  MoveL 8465 to (508.91, 504.67, 16.6) mm, rotated rx 0 ry 90 rz 0 deg; joints [-12.259, -27.847, 110.417, -16.319, -82.004, 51.311]
  Call Extruder(0.035)
  MoveL 8466 to (507.71, 504.67, 16.6) mm, rotated rx 0 ry 90 rz 0 deg; joints [-12.282, -27.872, 110.562, -16.338, -82.12, 51.279]
  Call Extruder(0.076)
  MoveL 8467 to (507.71, 502.07, 16.6) mm, rotated rx 0 ry 90 rz 0 deg; joints [-12.047, -27.883, 110.629, -16.098, -82.165, 51.235]
  Set speed (120.0 mm/s)
  MoveL 8468 to (508.03, 502.71, 16.6) mm, rotated rx 0 ry 90 rz 0 deg; joints [-12.099, -27.874, 110.575, -16.153, -82.124, 51.254]
  Set speed (15.0 mm/s)
  Call Extruder(0.014)
  MoveL 8469 to (508.36, 502.38, 16.6) mm, rotated rx 0 ry 90 rz 0 deg; joints [-12.063, -27.868, 110.544, -16.117, -82.098, 51.257]
  Set speed (120.0 mm/s)
  MoveL 8470 to (508.59, 503.13, 16.6) mm, rotated rx 0 ry 90 rz 0 deg; joints [-12.126, -27.86, 110.496, -16.183, -82.062, 51.276]
  Set speed (15.0 mm/s)
  Call Extruder(0.023)
  MoveL 8471 to (508.02, 503.7, 16.6) mm, rotated rx 0 ry 90 rz 0 deg; joints [-12.189, -27.869, 110.549, -16.244, -82.107, 51.271]
  Set speed (120.0 mm/s)
  MoveL 8472 to (508.59, 504.12, 16.6) mm, rotated rx 0 ry 90 rz 0 deg; joints [-12.216, -27.856, 110.47, -16.274, -82.044, 51.293]
  Set speed (15.0 mm/s)
  Call Extruder(0.010)
  MoveL 8473 to (508.36, 504.36, 16.6) mm, rotated rx 0 ry 90 rz 0 deg; joints [-12.241, -27.86, 110.492, -16.299, -82.063, 51.291]
  Set speed (120.0 mm/s)
  MoveL 8474 to (490.68, 490.68, 16.6) mm, rotated rx 0 ry 90 rz 0 deg; joints [-11.324, -28.243, 112.944, -15.306, -84.026, 50.625]
  Set speed (1000.0 mm/s)
  MoveL 8475 to (490.68, 490.68, 16.7) mm, rotated rx 0 ry 90 rz 0 deg; joints [-11.324, -28.254, 112.949, -15.306, -84.02, 50.627]
  Set speed (30.0 mm/s)
  Call Extruder(0.767)
  MoveL 8476 to (509.32, 509.32, 16.7) mm, rotated rx 0 ry 90 rz 0 deg; joints [-12.669, -27.828, 110.249, -16.739, -81.876, 51.405]
  MoveL 8477 to (509.44, 509.44, 16.7) mm, rotated rx 0 ry 90 rz 0 deg; joints [-12.677, -27.825, 110.231, -16.748, -81.862, 51.411]
  Set speed (120.0 mm/s)
  MoveL 8478 to (509.32, 500.58, 16.7) mm, rotated rx 0 ry 90 rz 0 deg; joints [-11.882, -27.867, 110.479, -15.937, -82.03, 51.252]
  Set speed (30.0 mm/s)
  Call Extruder(0.360)
  MoveL 8479 to (500.58, 509.32, 16.7) mm, rotated rx 0 ry 90 rz 0 deg; joints [-12.847, -28.002, 111.298, -16.885, -82.719, 51.172]
  Set speed (120.0 mm/s)
  MoveL 8480 to (499.42, 509.32, 16.7) mm, rotated rx 0 ry 90 rz 0 deg; joints [-12.872, -28.025, 111.436, -16.905, -82.831, 51.14]
  Set speed (30.0 mm/s)
  Call Extruder(0.360)
  MoveL 8481 to (490.68, 500.58, 16.7) mm, rotated rx 0 ry 90 rz 0 deg; joints [-12.247, -28.218, 112.705, -16.24, -83.843, 50.768]
  Set speed (120.0 mm/s)
  MoveL 8482 to (490.68, 499.42, 16.7) mm, rotated rx 0 ry 90 rz 0 deg; joints [-12.139, -28.223, 112.734, -16.131, -83.864, 50.751]
  Set speed (30.0 mm/s)
  MoveL 8483 to (499.42, 490.68, 16.7) mm, rotated rx 0 ry 90 rz 0 deg; joints [-11.163, -28.099, 111.91, -15.17, -83.162, 50.845]
  Set speed (120.0 mm/s)
  MoveL 8484 to (500.58, 490.68, 16.7) mm, rotated rx 0 ry 90 rz 0 deg; joints [-11.142, -28.077, 111.771, -15.153, -83.049, 50.874]
  Set speed (30.0 mm/s)
  MoveL 8485 to (509.32, 499.42, 16.7) mm, rotated rx 0 ry 90 rz 0 deg; joints [-11.777, -27.872, 110.508, -15.83, -82.05, 51.232]
  MoveL 8486 to (509.44, 499.54, 16.7) mm, rotated rx 0 ry 90 rz 0 deg; joints [-11.786, -27.869, 110.49, -15.84, -82.036, 51.237]
  Set speed (120.0 mm/s)
  MoveL 8487 to (509.32, 490.68, 16.7) mm, rotated rx 0 ry 90 rz 0 deg; joints [-10.985, -27.908, 110.72, -15.025, -82.193, 51.087]
  Set speed (30.0 mm/s)
  Call Extruder(0.767)
  MoveL 8488 to (490.68, 509.32, 16.7) mm, rotated rx 0 ry 90 rz 0 deg; joints [-13.056, -28.184, 112.473, -17.06, -83.676, 50.901]
  MoveL 8489 to (490.56, 509.44, 16.7) mm, rotated rx 0 ry 90 rz 0 deg; joints [-13.07, -28.186, 112.484, -17.074, -83.685, 50.9]
  Set speed (120.0 mm/s)
  MoveL 8490 to (490.4, 509.6, 16.7) mm, rotated rx 0 ry 90 rz 0 deg; joints [-13.088, -28.188, 112.498, -17.091, -83.697, 50.898]
  Set speed (15.0 mm/s)
  Call Extruder(0.559)
  MoveL 8491 to (490.4, 490.4, 16.7) mm, rotated rx 0 ry 90 rz 0 deg; joints [-11.303, -28.259, 112.989, -15.285, -84.052, 50.616]
  MoveL 8492 to (509.6, 490.4, 16.7) mm, rotated rx 0 ry 90 rz 0 deg; joints [-10.955, -27.903, 110.693, -14.995, -82.17, 51.089]
  MoveL 8493 to (509.6, 509.6, 16.7) mm, rotated rx 0 ry 90 rz 0 deg; joints [-12.688, -27.821, 110.208, -16.76, -81.844, 51.418]
  MoveL 8494 to (490.4, 509.6, 16.7) mm, rotated rx 0 ry 90 rz 0 deg; joints [-13.088, -28.188, 112.498, -17.091, -83.697, 50.898]
  Set speed (120.0 mm/s)
  MoveL 8495 to (490.4, 509.2, 16.7) mm, rotated rx 0 ry 90 rz 0 deg; joints [-13.051, -28.19, 112.509, -17.054, -83.705, 50.892]
  Set speed (1000.0 mm/s)
  MoveL 8496 to (490.5, 509.2, 16.7) mm, rotated rx 0 ry 90 rz 0 deg; joints [-13.049, -28.188, 112.497, -17.052, -83.696, 50.894]
  Set speed (1000.0 mm/s)
  MoveL 8497 to (494.92, 492.25, 16.7) mm, rotated rx 0 ry 90 rz 0 deg; joints [-11.391, -28.175, 112.409, -15.387, -83.577, 50.756]
  Set speed (15.0 mm/s)
  Call Extruder(0.034)
  MoveL 8498 to (494.92, 491.09, 16.7) mm, rotated rx 0 ry 90 rz 0 deg; joints [-11.283, -28.179, 112.436, -15.278, -83.597, 50.739]
  Call Extruder(0.071)
  MoveL 8499 to (497.34, 491.09, 16.7) mm, rotated rx 0 ry 90 rz 0 deg; joints [-11.238, -28.135, 112.147, -15.24, -83.359, 50.8]
  Call Extruder(0.034)
  MoveL 8500 to (497.34, 492.26, 16.7) mm, rotated rx 0 ry 90 rz 0 deg; joints [-11.347, -28.131, 112.12, -15.35, -83.339, 50.817]
  Call Extruder(0.069)
  MoveL 8501 to (494.97, 492.26, 16.7) mm, rotated rx 0 ry 90 rz 0 deg; joints [-11.391, -28.174, 112.402, -15.387, -83.571, 50.757]
  Call Extruder(0.000)
  MoveL 8502 to (494.97, 492.25, 16.7) mm, rotated rx 0 ry 90 rz 0 deg; joints [-11.39, -28.174, 112.402, -15.387, -83.572, 50.757]
  Call Extruder(0.002)
  MoveL 8503 to (494.92, 492.25, 16.7) mm, rotated rx 0 ry 90 rz 0 deg; joints [-11.391, -28.175, 112.409, -15.387, -83.577, 50.756]
  Set speed (120.0 mm/s)
  MoveL 8504 to (495.36, 491.4, 16.7) mm, rotated rx 0 ry 90 rz 0 deg; joints [-11.304, -28.17, 112.376, -15.301, -83.548, 50.755]
  Set speed (15.0 mm/s)
  Call Extruder(0.022)
  MoveL 8505 to (495.91, 491.95, 16.7) mm, rotated rx 0 ry 90 rz 0 deg; joints [-11.344, -28.158, 112.298, -15.343, -83.485, 50.776]
  Set speed (120.0 mm/s)
  MoveL 8506 to (496.35, 491.4, 16.7) mm, rotated rx 0 ry 90 rz 0 deg; joints [-11.286, -28.152, 112.258, -15.285, -83.451, 50.779]
  Set speed (15.0 mm/s)
  MoveL 8507 to (496.9, 491.95, 16.7) mm, rotated rx 0 ry 90 rz 0 deg; joints [-11.326, -28.14, 112.181, -15.328, -83.388, 50.801]
  Set speed (120.0 mm/s)
  MoveL 8508 to (502.03, 492.26, 16.7) mm, rotated rx 0 ry 90 rz 0 deg; joints [-11.261, -28.044, 111.56, -15.279, -82.881, 50.933]
  Set speed (15.0 mm/s)
  Call Extruder(0.034)
  MoveL 8509 to (502.03, 491.09, 16.7) mm, rotated rx 0 ry 90 rz 0 deg; joints [-11.153, -28.049, 111.588, -15.169, -82.9, 50.915]
  Call Extruder(0.071)
  MoveL 8510 to (504.46, 491.09, 16.7) mm, rotated rx 0 ry 90 rz 0 deg; joints [-11.109, -28.002, 111.296, -15.133, -82.662, 50.975]
  Call Extruder(0.034)
  MoveL 8511 to (504.46, 492.27, 16.7) mm, rotated rx 0 ry 90 rz 0 deg; joints [-11.217, -27.998, 111.268, -15.243, -82.643, 50.994]
  Call Extruder(0.016)
  MoveL 8512 to (503.92, 492.26, 16.7) mm, rotated rx 0 ry 90 rz 0 deg; joints [-11.226, -28.008, 111.333, -15.25, -82.695, 50.98]
  Call Extruder(0.055)
  MoveL 8513 to (502.03, 492.26, 16.7) mm, rotated rx 0 ry 90 rz 0 deg; joints [-11.261, -28.044, 111.56, -15.279, -82.881, 50.933]
  Set speed (120.0 mm/s)
  MoveL 8514 to (502.84, 491.95, 16.7) mm, rotated rx 0 ry 90 rz 0 deg; joints [-11.217, -28.03, 111.471, -15.237, -82.807, 50.949]
  Set speed (15.0 mm/s)
  Call Extruder(0.020)
  MoveL 8515 to (502.34, 491.45, 16.7) mm, rotated rx 0 ry 90 rz 0 deg; joints [-11.18, -28.041, 111.542, -15.198, -82.864, 50.929]
  Set speed (120.0 mm/s)
  MoveL 8516 to (503.28, 491.41, 16.7) mm, rotated rx 0 ry 90 rz 0 deg; joints [-11.159, -28.024, 111.43, -15.18, -82.772, 50.951]
  Set speed (15.0 mm/s)
  Call Extruder(0.022)
  MoveL 8517 to (503.83, 491.95, 16.7) mm, rotated rx 0 ry 90 rz 0 deg; joints [-11.199, -28.011, 111.352, -15.222, -82.71, 50.973]
  Set speed (120.0 mm/s)
  MoveL 8518 to (507.71, 494.38, 16.7) mm, rotated rx 0 ry 90 rz 0 deg; joints [-11.351, -27.925, 110.826, -15.39, -82.29, 51.108]
  Set speed (15.0 mm/s)
  Call Extruder(0.035)
  MoveL 8519 to (508.91, 494.38, 16.7) mm, rotated rx 0 ry 90 rz 0 deg; joints [-11.328, -27.901, 110.682, -15.372, -82.174, 51.137]
  Call Extruder(0.074)
  MoveL 8520 to (508.91, 496.9, 16.7) mm, rotated rx 0 ry 90 rz 0 deg; joints [-11.557, -27.891, 110.62, -15.605, -82.132, 51.179]
  Call Extruder(0.035)
  MoveL 8521 to (507.71, 496.9, 16.7) mm, rotated rx 0 ry 90 rz 0 deg; joints [-11.579, -27.915, 110.764, -15.623, -82.248, 51.149]
  Call Extruder(0.051)
  MoveL 8522 to (507.72, 495.15, 16.7) mm, rotated rx 0 ry 90 rz 0 deg; joints [-11.42, -27.922, 110.807, -15.461, -82.277, 51.12]
  Call Extruder(0.022)
  MoveL 8523 to (507.71, 494.38, 16.7) mm, rotated rx 0 ry 90 rz 0 deg; joints [-11.351, -27.925, 110.826, -15.39, -82.29, 51.108]
  Set speed (120.0 mm/s)
  MoveL 8524 to (508.03, 495.16, 16.7) mm, rotated rx 0 ry 90 rz 0 deg; joints [-11.415, -27.916, 110.769, -15.457, -82.247, 51.128]
  Set speed (15.0 mm/s)
  Call Extruder(0.023)
  MoveL 8525 to (508.59, 495.72, 16.7) mm, rotated rx 0 ry 90 rz 0 deg; joints [-11.456, -27.902, 110.687, -15.501, -82.182, 51.152]
  Set speed (120.0 mm/s)
  MoveL 8526 to (508.03, 496.15, 16.7) mm, rotated rx 0 ry 90 rz 0 deg; joints [-11.505, -27.912, 110.745, -15.548, -82.23, 51.145]
  Set speed (15.0 mm/s)
  Call Extruder(0.018)
  MoveL 8527 to (508.46, 496.59, 16.7) mm, rotated rx 0 ry 90 rz 0 deg; joints [-11.537, -27.901, 110.681, -15.582, -82.18, 51.163]
  Set speed (120.0 mm/s)
  MoveL 8528 to (508.91, 502.12, 16.7) mm, rotated rx 0 ry 90 rz 0 deg; joints [-12.029, -27.869, 110.489, -16.085, -82.043, 51.268]
  Set speed (15.0 mm/s)
  Call Extruder(0.074)
  MoveL 8529 to (508.91, 504.67, 16.7) mm, rotated rx 0 ry 90 rz 0 deg; joints [-12.259, -27.858, 110.422, -16.319, -81.999, 51.312]
  Call Extruder(0.035)
  MoveL 8530 to (507.71, 504.67, 16.7) mm, rotated rx 0 ry 90 rz 0 deg; joints [-12.282, -27.882, 110.567, -16.338, -82.115, 51.281]
  Call Extruder(0.074)
  MoveL 8531 to (507.71, 502.12, 16.7) mm, rotated rx 0 ry 90 rz 0 deg; joints [-12.052, -27.893, 110.633, -16.104, -82.159, 51.237]
  Call Extruder(0.035)
  MoveL 8532 to (508.91, 502.12, 16.7) mm, rotated rx 0 ry 90 rz 0 deg; joints [-12.029, -27.869, 110.489, -16.085, -82.043, 51.268]
  Set speed (120.0 mm/s)
  MoveL 8533 to (508.59, 502.65, 16.7) mm, rotated rx 0 ry 90 rz 0 deg; joints [-12.083, -27.873, 110.513, -16.139, -82.065, 51.269]
  Set speed (15.0 mm/s)
  Call Extruder(0.009)
  MoveL 8534 to (508.38, 502.44, 16.7) mm, rotated rx 0 ry 90 rz 0 deg; joints [-12.068, -27.878, 110.545, -16.122, -82.089, 51.26]
  Set speed (120.0 mm/s)
  MoveL 8535 to (508.03, 503.08, 16.7) mm, rotated rx 0 ry 90 rz 0 deg; joints [-12.132, -27.883, 110.571, -16.187, -82.112, 51.261]
  Set speed (15.0 mm/s)
  Call Extruder(0.023)
  MoveL 8536 to (508.59, 503.64, 16.7) mm, rotated rx 0 ry 90 rz 0 deg; joints [-12.172, -27.869, 110.487, -16.23, -82.047, 51.286]
  Set speed (120.0 mm/s)
  MoveL 8537 to (508.02, 504.06, 16.7) mm, rotated rx 0 ry 90 rz 0 deg; joints [-12.221, -27.878, 110.545, -16.277, -82.095, 51.278]
  Set speed (15.0 mm/s)
  Call Extruder(0.012)
  MoveL 8538 to (508.32, 504.36, 16.7) mm, rotated rx 0 ry 90 rz 0 deg; joints [-12.242, -27.871, 110.502, -16.3, -82.062, 51.291]
  Set speed (120.0 mm/s)
  MoveL 8539 to (490.68, 490.68, 16.7) mm, rotated rx 0 ry 90 rz 0 deg; joints [-11.324, -28.254, 112.949, -15.306, -84.02, 50.627]
  Set speed (1000.0 mm/s)
  MoveL 8540 to (490.68, 490.68, 16.8) mm, rotated rx 0 ry 90 rz 0 deg; joints [-11.324, -28.264, 112.954, -15.307, -84.015, 50.628]
  Set speed (30.0 mm/s)
  Call Extruder(0.767)
  MoveL 8541 to (509.32, 509.32, 16.8) mm, rotated rx 0 ry 90 rz 0 deg; joints [-12.669, -27.838, 110.254, -16.739, -81.871, 51.407]
  MoveL 8542 to (509.44, 509.44, 16.8) mm, rotated rx 0 ry 90 rz 0 deg; joints [-12.677, -27.835, 110.236, -16.748, -81.857, 51.412]
  Set speed (120.0 mm/s)
  MoveL 8543 to (509.32, 500.58, 16.8) mm, rotated rx 0 ry 90 rz 0 deg; joints [-11.882, -27.878, 110.484, -15.937, -82.025, 51.253]
  Set speed (30.0 mm/s)
  Call Extruder(0.360)
  MoveL 8544 to (500.58, 509.32, 16.8) mm, rotated rx 0 ry 90 rz 0 deg; joints [-12.847, -28.013, 111.303, -16.885, -82.714, 51.173]
  Set speed (120.0 mm/s)
  MoveL 8545 to (499.42, 509.32, 16.8) mm, rotated rx 0 ry 90 rz 0 deg; joints [-12.872, -28.035, 111.441, -16.905, -82.826, 51.142]
  Set speed (30.0 mm/s)
  Call Extruder(0.360)
  MoveL 8546 to (490.68, 500.58, 16.8) mm, rotated rx 0 ry 90 rz 0 deg; joints [-12.247, -28.229, 112.71, -16.24, -83.837, 50.77]
  Set speed (120.0 mm/s)
  MoveL 8547 to (490.68, 499.42, 16.8) mm, rotated rx 0 ry 90 rz 0 deg; joints [-12.139, -28.233, 112.739, -16.131, -83.859, 50.752]
  Set speed (30.0 mm/s)
  MoveL 8548 to (499.42, 490.68, 16.8) mm, rotated rx 0 ry 90 rz 0 deg; joints [-11.163, -28.11, 111.915, -15.17, -83.157, 50.846]
  Set speed (120.0 mm/s)
  MoveL 8549 to (500.58, 490.68, 16.8) mm, rotated rx 0 ry 90 rz 0 deg; joints [-11.141, -28.088, 111.776, -15.153, -83.043, 50.875]
  Set speed (30.0 mm/s)
  MoveL 8550 to (509.32, 499.42, 16.8) mm, rotated rx 0 ry 90 rz 0 deg; joints [-11.777, -27.883, 110.513, -15.831, -82.045, 51.233]
  MoveL 8551 to (509.44, 499.54, 16.8) mm, rotated rx 0 ry 90 rz 0 deg; joints [-11.786, -27.879, 110.495, -15.84, -82.031, 51.239]
  Set speed (120.0 mm/s)
  MoveL 8552 to (509.32, 490.68, 16.8) mm, rotated rx 0 ry 90 rz 0 deg; joints [-10.985, -27.918, 110.725, -15.025, -82.188, 51.088]
  Set speed (30.0 mm/s)
  Call Extruder(0.767)
  MoveL 8553 to (490.68, 509.32, 16.8) mm, rotated rx 0 ry 90 rz 0 deg; joints [-13.056, -28.195, 112.478, -17.06, -83.671, 50.903]
  MoveL 8554 to (490.56, 509.44, 16.8) mm, rotated rx 0 ry 90 rz 0 deg; joints [-13.07, -28.197, 112.489, -17.074, -83.68, 50.901]
  Set speed (120.0 mm/s)
  MoveL 8555 to (490.4, 509.6, 16.8) mm, rotated rx 0 ry 90 rz 0 deg; joints [-13.088, -28.199, 112.503, -17.092, -83.692, 50.9]
  Set speed (15.0 mm/s)
  Call Extruder(0.559)
  MoveL 8556 to (490.4, 490.4, 16.8) mm, rotated rx 0 ry 90 rz 0 deg; joints [-11.303, -28.27, 112.994, -15.285, -84.047, 50.617]
  MoveL 8557 to (509.6, 490.4, 16.8) mm, rotated rx 0 ry 90 rz 0 deg; joints [-10.955, -27.914, 110.698, -14.995, -82.165, 51.091]
  MoveL 8558 to (509.6, 509.6, 16.8) mm, rotated rx 0 ry 90 rz 0 deg; joints [-12.688, -27.831, 110.213, -16.76, -81.839, 51.419]
  MoveL 8559 to (490.4, 509.6, 16.8) mm, rotated rx 0 ry 90 rz 0 deg; joints [-13.088, -28.199, 112.503, -17.092, -83.692, 50.9]
  Set speed (120.0 mm/s)
  MoveL 8560 to (490.4, 509.2, 16.8) mm, rotated rx 0 ry 90 rz 0 deg; joints [-13.051, -28.2, 112.514, -17.054, -83.7, 50.893]
  Set speed (1000.0 mm/s)
  MoveL 8561 to (490.5, 509.2, 16.8) mm, rotated rx 0 ry 90 rz 0 deg; joints [-13.049, -28.199, 112.502, -17.052, -83.69, 50.896]
  Set speed (1000.0 mm/s)
  MoveL 8562 to (494.92, 492.25, 16.8) mm, rotated rx 0 ry 90 rz 0 deg; joints [-11.391, -28.185, 112.414, -15.387, -83.572, 50.757]
  Set speed (15.0 mm/s)
  Call Extruder(0.034)
  MoveL 8563 to (494.92, 491.09, 16.8) mm, rotated rx 0 ry 90 rz 0 deg; joints [-11.283, -28.19, 112.442, -15.278, -83.592, 50.74]
  Call Extruder(0.069)
  MoveL 8564 to (497.28, 491.09, 16.8) mm, rotated rx 0 ry 90 rz 0 deg; joints [-11.24, -28.147, 112.16, -15.242, -83.36, 50.799]
  Call Extruder(0.034)
  MoveL 8565 to (497.27, 492.27, 16.8) mm, rotated rx 0 ry 90 rz 0 deg; joints [-11.348, -28.143, 112.133, -15.352, -83.341, 50.817]
  Call Extruder(0.069)
  MoveL 8566 to (494.92, 492.25, 16.8) mm, rotated rx 0 ry 90 rz 0 deg; joints [-11.391, -28.185, 112.414, -15.387, -83.572, 50.757]
  Set speed (120.0 mm/s)
  MoveL 8567 to (495.23, 491.75, 16.8) mm, rotated rx 0 ry 90 rz 0 deg; joints [-11.339, -28.182, 112.389, -15.335, -83.55, 50.758]
  Set speed (15.0 mm/s)
  Call Extruder(0.014)
  MoveL 8568 to (495.57, 491.4, 16.8) mm, rotated rx 0 ry 90 rz 0 deg; joints [-11.3, -28.177, 112.356, -15.298, -83.522, 50.761]
  Set speed (120.0 mm/s)
  MoveL 8569 to (496.03, 491.94, 16.8) mm, rotated rx 0 ry 90 rz 0 deg; joints [-11.342, -28.167, 112.289, -15.341, -83.468, 50.781]
  Set speed (15.0 mm/s)
  Call Extruder(0.022)
  MoveL 8570 to (496.57, 491.4, 16.8) mm, rotated rx 0 ry 90 rz 0 deg; joints [-11.282, -28.159, 112.238, -15.282, -83.425, 50.786]
  Set speed (120.0 mm/s)
  MoveL 8571 to (502.09, 491.09, 16.8) mm, rotated rx 0 ry 90 rz 0 deg; joints [-11.152, -28.058, 111.586, -15.169, -82.889, 50.918]
  Set speed (15.0 mm/s)
  Call Extruder(0.069)
  MoveL 8572 to (504.46, 491.09, 16.8) mm, rotated rx 0 ry 90 rz 0 deg; joints [-11.109, -28.013, 111.301, -15.133, -82.657, 50.977]
  Call Extruder(0.034)
  MoveL 8573 to (504.46, 492.27, 16.8) mm, rotated rx 0 ry 90 rz 0 deg; joints [-11.217, -28.008, 111.273, -15.243, -82.638, 50.995]
  Call Extruder(0.069)
  MoveL 8574 to (502.09, 492.24, 16.8) mm, rotated rx 0 ry 90 rz 0 deg; joints [-11.258, -28.054, 111.558, -15.276, -82.87, 50.936]
  Call Extruder(0.034)
  MoveL 8575 to (502.09, 491.09, 16.8) mm, rotated rx 0 ry 90 rz 0 deg; joints [-11.152, -28.058, 111.586, -15.169, -82.889, 50.918]
  Set speed (120.0 mm/s)
  MoveL 8576 to (502.4, 491.51, 16.8) mm, rotated rx 0 ry 90 rz 0 deg; joints [-11.184, -28.051, 111.538, -15.203, -82.851, 50.933]
  Set speed (15.0 mm/s)
  Call Extruder(0.004)
  MoveL 8577 to (502.5, 491.4, 16.8) mm, rotated rx 0 ry 90 rz 0 deg; joints [-11.173, -28.049, 111.528, -15.192, -82.843, 50.934]
  Set speed (120.0 mm/s)
  MoveL 8578 to (502.96, 491.94, 16.8) mm, rotated rx 0 ry 90 rz 0 deg; joints [-11.214, -28.038, 111.461, -15.234, -82.789, 50.953]
  Set speed (15.0 mm/s)
  Call Extruder(0.022)
  MoveL 8579 to (503.49, 491.4, 16.8) mm, rotated rx 0 ry 90 rz 0 deg; joints [-11.155, -28.03, 111.41, -15.177, -82.746, 50.958]
  Set speed (120.0 mm/s)
  MoveL 8580 to (503.94, 491.95, 16.8) mm, rotated rx 0 ry 90 rz 0 deg; joints [-11.197, -28.019, 111.343, -15.221, -82.693, 50.977]
  Set speed (15.0 mm/s)
  Call Extruder(0.008)
  MoveL 8581 to (504.14, 491.75, 16.8) mm, rotated rx 0 ry 90 rz 0 deg; joints [-11.175, -28.016, 111.324, -15.199, -82.677, 50.979]
  Set speed (120.0 mm/s)
  MoveL 8582 to (507.72, 494.39, 16.8) mm, rotated rx 0 ry 90 rz 0 deg; joints [-11.351, -27.936, 110.831, -15.391, -82.285, 51.109]
  Set speed (15.0 mm/s)
  Call Extruder(0.035)
  MoveL 8583 to (508.91, 494.38, 16.8) mm, rotated rx 0 ry 90 rz 0 deg; joints [-11.328, -27.912, 110.687, -15.372, -82.168, 51.139]
  Call Extruder(0.072)
  MoveL 8584 to (508.91, 496.84, 16.8) mm, rotated rx 0 ry 90 rz 0 deg; joints [-11.551, -27.902, 110.627, -15.599, -82.128, 51.18]
  Call Extruder(0.035)
  MoveL 8585 to (507.71, 496.83, 16.8) mm, rotated rx 0 ry 90 rz 0 deg; joints [-11.573, -27.926, 110.771, -15.617, -82.244, 51.15]
  Call Extruder(0.071)
  MoveL 8586 to (507.72, 494.39, 16.8) mm, rotated rx 0 ry 90 rz 0 deg; joints [-11.351, -27.936, 110.831, -15.391, -82.285, 51.109]
  Set speed (120.0 mm/s)
  MoveL 8587 to (508.59, 495.21, 16.8) mm, rotated rx 0 ry 90 rz 0 deg; joints [-11.41, -27.915, 110.705, -15.454, -82.185, 51.145]
  Set speed (15.0 mm/s)
  Call Extruder(0.023)
  MoveL 8588 to (508.03, 495.78, 16.8) mm, rotated rx 0 ry 90 rz 0 deg; joints [-11.472, -27.924, 110.759, -15.515, -82.231, 51.14]
  Set speed (120.0 mm/s)
  MoveL 8589 to (508.59, 496.2, 16.8) mm, rotated rx 0 ry 90 rz 0 deg; joints [-11.5, -27.911, 110.68, -15.545, -82.169, 51.161]
  Set speed (15.0 mm/s)
  Call Extruder(0.013)
  MoveL 8590 to (508.28, 496.52, 16.8) mm, rotated rx 0 ry 90 rz 0 deg; joints [-11.534, -27.916, 110.711, -15.579, -82.195, 51.159]
  Set speed (120.0 mm/s)
  MoveL 8591 to (507.71, 502.18, 16.8) mm, rotated rx 0 ry 90 rz 0 deg; joints [-12.057, -27.903, 110.637, -16.109, -82.153, 51.24]
  Set speed (15.0 mm/s)
  Call Extruder(0.035)
  MoveL 8592 to (508.91, 502.18, 16.8) mm, rotated rx 0 ry 90 rz 0 deg; joints [-12.034, -27.879, 110.492, -16.09, -82.037, 51.27]
  Call Extruder(0.073)
  MoveL 8593 to (508.91, 504.67, 16.8) mm, rotated rx 0 ry 90 rz 0 deg; joints [-12.259, -27.868, 110.427, -16.32, -81.993, 51.314]
  Call Extruder(0.035)
  MoveL 8594 to (507.71, 504.67, 16.8) mm, rotated rx 0 ry 90 rz 0 deg; joints [-12.282, -27.892, 110.572, -16.339, -82.11, 51.282]
  Call Extruder(0.073)
  MoveL 8595 to (507.71, 502.18, 16.8) mm, rotated rx 0 ry 90 rz 0 deg; joints [-12.057, -27.903, 110.637, -16.109, -82.153, 51.24]
  Set speed (120.0 mm/s)
  MoveL 8596 to (508.25, 502.49, 16.8) mm, rotated rx 0 ry 90 rz 0 deg; joints [-12.075, -27.891, 110.564, -16.13, -82.096, 51.259]
  Set speed (15.0 mm/s)
  Call Extruder(0.009)
  MoveL 8597 to (508.03, 502.71, 16.8) mm, rotated rx 0 ry 90 rz 0 deg; joints [-12.099, -27.895, 110.585, -16.153, -82.113, 51.257]
  Set speed (120.0 mm/s)
  MoveL 8598 to (508.59, 503.13, 16.8) mm, rotated rx 0 ry 90 rz 0 deg; joints [-12.126, -27.881, 110.506, -16.183, -82.051, 51.279]
  Set speed (15.0 mm/s)
  Call Extruder(0.023)
  MoveL 8599 to (508.02, 503.7, 16.8) mm, rotated rx 0 ry 90 rz 0 deg; joints [-12.189, -27.89, 110.559, -16.244, -82.096, 51.274]
  Set speed (120.0 mm/s)
  MoveL 8600 to (508.59, 504.12, 16.8) mm, rotated rx 0 ry 90 rz 0 deg; joints [-12.216, -27.877, 110.48, -16.274, -82.034, 51.296]
  Set speed (15.0 mm/s)
  Call Extruder(0.010)
  MoveL 8601 to (508.36, 504.36, 16.8) mm, rotated rx 0 ry 90 rz 0 deg; joints [-12.241, -27.881, 110.502, -16.299, -82.052, 51.294]
  Set speed (120.0 mm/s)
  MoveL 8602 to (490.68, 490.68, 16.8) mm, rotated rx 0 ry 90 rz 0 deg; joints [-11.324, -28.264, 112.954, -15.307, -84.015, 50.628]
  Set speed (1000.0 mm/s)
  MoveL 8603 to (490.68, 490.68, 16.9) mm, rotated rx 0 ry 90 rz 0 deg; joints [-11.324, -28.275, 112.959, -15.307, -84.009, 50.63]
  Set speed (30.0 mm/s)
  Call Extruder(0.767)
  MoveL 8604 to (509.32, 509.32, 16.9) mm, rotated rx 0 ry 90 rz 0 deg; joints [-12.669, -27.849, 110.259, -16.739, -81.866, 51.408]
  MoveL 8605 to (509.44, 509.44, 16.9) mm, rotated rx 0 ry 90 rz 0 deg; joints [-12.677, -27.846, 110.241, -16.748, -81.852, 51.414]
  Set speed (120.0 mm/s)
  MoveL 8606 to (509.32, 500.58, 16.9) mm, rotated rx 0 ry 90 rz 0 deg; joints [-11.882, -27.888, 110.489, -15.937, -82.02, 51.255]
  Set speed (30.0 mm/s)
  Call Extruder(0.360)
  MoveL 8607 to (500.58, 509.32, 16.9) mm, rotated rx 0 ry 90 rz 0 deg; joints [-12.847, -28.023, 111.308, -16.885, -82.709, 51.175]
  Set speed (120.0 mm/s)
  MoveL 8608 to (499.42, 509.32, 16.9) mm, rotated rx 0 ry 90 rz 0 deg; joints [-12.872, -28.046, 111.446, -16.905, -82.821, 51.143]
  Set speed (30.0 mm/s)
  Call Extruder(0.360)
  MoveL 8609 to (490.68, 500.58, 16.9) mm, rotated rx 0 ry 90 rz 0 deg; joints [-12.247, -28.24, 112.715, -16.24, -83.832, 50.771]
  Set speed (120.0 mm/s)
  MoveL 8610 to (490.68, 499.42, 16.9) mm, rotated rx 0 ry 90 rz 0 deg; joints [-12.139, -28.244, 112.745, -16.131, -83.853, 50.754]
  Set speed (30.0 mm/s)
  MoveL 8611 to (499.42, 490.68, 16.9) mm, rotated rx 0 ry 90 rz 0 deg; joints [-11.163, -28.12, 111.92, -15.171, -83.152, 50.848]
  Set speed (120.0 mm/s)
  MoveL 8612 to (500.58, 490.68, 16.9) mm, rotated rx 0 ry 90 rz 0 deg; joints [-11.141, -28.099, 111.781, -15.153, -83.038, 50.876]
  Set speed (30.0 mm/s)
  MoveL 8613 to (509.32, 499.42, 16.9) mm, rotated rx 0 ry 90 rz 0 deg; joints [-11.777, -27.893, 110.518, -15.831, -82.039, 51.235]
  MoveL 8614 to (509.44, 499.54, 16.9) mm, rotated rx 0 ry 90 rz 0 deg; joints [-11.786, -27.89, 110.5, -15.84, -82.025, 51.24]
  Set speed (120.0 mm/s)
  MoveL 8615 to (509.32, 490.68, 16.9) mm, rotated rx 0 ry 90 rz 0 deg; joints [-10.985, -27.929, 110.73, -15.025, -82.183, 51.09]
  Set speed (30.0 mm/s)
  Call Extruder(0.767)
  MoveL 8616 to (490.68, 509.32, 16.9) mm, rotated rx 0 ry 90 rz 0 deg; joints [-13.056, -28.206, 112.483, -17.06, -83.665, 50.905]
  MoveL 8617 to (490.56, 509.44, 16.9) mm, rotated rx 0 ry 90 rz 0 deg; joints [-13.07, -28.207, 112.494, -17.074, -83.675, 50.903]
  Set speed (120.0 mm/s)
  MoveL 8618 to (490.4, 509.6, 16.9) mm, rotated rx 0 ry 90 rz 0 deg; joints [-13.088, -28.209, 112.508, -17.092, -83.687, 50.901]
  Set speed (15.0 mm/s)
  Call Extruder(0.559)
  MoveL 8619 to (490.4, 490.4, 16.9) mm, rotated rx 0 ry 90 rz 0 deg; joints [-11.303, -28.281, 112.999, -15.285, -84.042, 50.619]
  MoveL 8620 to (509.6, 490.4, 16.9) mm, rotated rx 0 ry 90 rz 0 deg; joints [-10.955, -27.924, 110.703, -14.996, -82.16, 51.092]
  MoveL 8621 to (509.6, 509.6, 16.9) mm, rotated rx 0 ry 90 rz 0 deg; joints [-12.688, -27.842, 110.218, -16.76, -81.834, 51.421]
  MoveL 8622 to (490.4, 509.6, 16.9) mm, rotated rx 0 ry 90 rz 0 deg; joints [-13.088, -28.209, 112.508, -17.092, -83.687, 50.901]
  Set speed (120.0 mm/s)
  MoveL 8623 to (490.4, 509.2, 16.9) mm, rotated rx 0 ry 90 rz 0 deg; joints [-13.051, -28.211, 112.519, -17.054, -83.695, 50.895]
  Set speed (1000.0 mm/s)
  MoveL 8624 to (490.5, 509.2, 16.9) mm, rotated rx 0 ry 90 rz 0 deg; joints [-13.049, -28.209, 112.507, -17.052, -83.685, 50.898]
  Set speed (1000.0 mm/s)
  MoveL 8625 to (507.71, 504.67, 16.9) mm, rotated rx 0 ry 90 rz 0 deg; joints [-12.282, -27.903, 110.577, -16.339, -82.104, 51.284]
  Set speed (15.0 mm/s)
  Call Extruder(0.071)
  MoveL 8626 to (507.71, 502.23, 16.9) mm, rotated rx 0 ry 90 rz 0 deg; joints [-12.062, -27.914, 110.64, -16.114, -82.147, 51.242]
  Call Extruder(0.035)
  MoveL 8627 to (508.91, 502.23, 16.9) mm, rotated rx 0 ry 90 rz 0 deg; joints [-12.039, -27.889, 110.496, -16.096, -82.031, 51.273]
  Call Extruder(0.071)
  MoveL 8628 to (508.91, 504.67, 16.9) mm, rotated rx 0 ry 90 rz 0 deg; joints [-12.259, -27.878, 110.432, -16.32, -81.988, 51.315]
  Call Extruder(0.035)
  MoveL 8629 to (507.71, 504.67, 16.9) mm, rotated rx 0 ry 90 rz 0 deg; joints [-12.282, -27.903, 110.577, -16.339, -82.104, 51.284]
  Set speed (120.0 mm/s)
  MoveL 8630 to (508.32, 504.36, 16.9) mm, rotated rx 0 ry 90 rz 0 deg; joints [-12.242, -27.892, 110.512, -16.3, -82.051, 51.294]
  Set speed (15.0 mm/s)
  Call Extruder(0.012)
  MoveL 8631 to (508.02, 504.06, 16.9) mm, rotated rx 0 ry 90 rz 0 deg; joints [-12.221, -27.899, 110.555, -16.278, -82.085, 51.282]
  Set speed (120.0 mm/s)
  MoveL 8632 to (508.59, 503.64, 16.9) mm, rotated rx 0 ry 90 rz 0 deg; joints [-12.172, -27.89, 110.497, -16.23, -82.037, 51.289]
  Set speed (15.0 mm/s)
  Call Extruder(0.023)
  MoveL 8633 to (508.02, 503.08, 16.9) mm, rotated rx 0 ry 90 rz 0 deg; joints [-12.132, -27.904, 110.581, -16.187, -82.102, 51.265]
  Set speed (120.0 mm/s)
  MoveL 8634 to (508.49, 502.55, 16.9) mm, rotated rx 0 ry 90 rz 0 deg; joints [-12.076, -27.896, 110.539, -16.131, -82.066, 51.267]
  Set speed (15.0 mm/s)
  Call Extruder(0.004)
  MoveL 8635 to (508.59, 502.65, 16.9) mm, rotated rx 0 ry 90 rz 0 deg; joints [-12.083, -27.894, 110.523, -16.139, -82.054, 51.272]
  Set speed (120.0 mm/s)
  MoveL 8636 to (490.68, 490.68, 16.9) mm, rotated rx 0 ry 90 rz 0 deg; joints [-11.324, -28.275, 112.959, -15.307, -84.009, 50.63]
  Set speed (1000.0 mm/s)
  MoveL 8637 to (490.68, 490.68, 17) mm, rotated rx 0 ry 90 rz 0 deg; joints [-11.324, -28.286, 112.964, -15.307, -84.004, 50.631]
  Set speed (30.0 mm/s)
  Call Extruder(0.767)
  MoveL 8638 to (509.32, 509.32, 17) mm, rotated rx 0 ry 90 rz 0 deg; joints [-12.669, -27.859, 110.265, -16.739, -81.861, 51.41]
  MoveL 8639 to (509.44, 509.44, 17) mm, rotated rx 0 ry 90 rz 0 deg; joints [-12.677, -27.856, 110.246, -16.748, -81.847, 51.415]
  Set speed (120.0 mm/s)
  MoveL 8640 to (509.32, 500.58, 17) mm, rotated rx 0 ry 90 rz 0 deg; joints [-11.882, -27.899, 110.494, -15.938, -82.014, 51.256]
  Set speed (30.0 mm/s)
  Call Extruder(0.360)
  MoveL 8641 to (500.58, 509.32, 17) mm, rotated rx 0 ry 90 rz 0 deg; joints [-12.847, -28.034, 111.313, -16.885, -82.704, 51.176]
  Set speed (120.0 mm/s)
  MoveL 8642 to (499.42, 509.32, 17) mm, rotated rx 0 ry 90 rz 0 deg; joints [-12.872, -28.056, 111.451, -16.905, -82.815, 51.145]
  Set speed (30.0 mm/s)
  Call Extruder(0.360)
  MoveL 8643 to (490.68, 500.58, 17) mm, rotated rx 0 ry 90 rz 0 deg; joints [-12.247, -28.25, 112.72, -16.241, -83.827, 50.773]
  Set speed (120.0 mm/s)
  MoveL 8644 to (490.68, 499.42, 17) mm, rotated rx 0 ry 90 rz 0 deg; joints [-12.139, -28.255, 112.75, -16.131, -83.848, 50.756]
  Set speed (30.0 mm/s)
  MoveL 8645 to (499.42, 490.68, 17) mm, rotated rx 0 ry 90 rz 0 deg; joints [-11.163, -28.131, 111.925, -15.171, -83.146, 50.849]
  Set speed (120.0 mm/s)
  MoveL 8646 to (500.58, 490.68, 17) mm, rotated rx 0 ry 90 rz 0 deg; joints [-11.141, -28.109, 111.786, -15.153, -83.033, 50.878]
  Set speed (30.0 mm/s)
  Call Extruder(0.360)
  MoveL 8647 to (509.32, 499.42, 17) mm, rotated rx 0 ry 90 rz 0 deg; joints [-11.777, -27.903, 110.523, -15.831, -82.034, 51.236]
  MoveL 8648 to (509.44, 499.54, 17) mm, rotated rx 0 ry 90 rz 0 deg; joints [-11.786, -27.9, 110.505, -15.841, -82.02, 51.242]
  Set speed (120.0 mm/s)
  MoveL 8649 to (509.32, 490.68, 17) mm, rotated rx 0 ry 90 rz 0 deg; joints [-10.985, -27.939, 110.736, -15.026, -82.178, 51.091]
  Set speed (30.0 mm/s)
  Call Extruder(0.767)
  MoveL 8650 to (490.68, 509.32, 17) mm, rotated rx 0 ry 90 rz 0 deg; joints [-13.056, -28.216, 112.488, -17.061, -83.66, 50.906]
  MoveL 8651 to (490.56, 509.44, 17) mm, rotated rx 0 ry 90 rz 0 deg; joints [-13.07, -28.218, 112.499, -17.074, -83.67, 50.905]
  Set speed (120.0 mm/s)
  MoveL 8652 to (490.4, 509.6, 17) mm, rotated rx 0 ry 90 rz 0 deg; joints [-13.088, -28.22, 112.513, -17.092, -83.682, 50.903]
  Set speed (15.0 mm/s)
  Call Extruder(0.559)
  MoveL 8653 to (490.4, 490.4, 17) mm, rotated rx 0 ry 90 rz 0 deg; joints [-11.303, -28.292, 113.004, -15.285, -84.036, 50.62]
  MoveL 8654 to (509.6, 490.4, 17) mm, rotated rx 0 ry 90 rz 0 deg; joints [-10.955, -27.935, 110.708, -14.996, -82.155, 51.093]
  MoveL 8655 to (509.6, 509.6, 17) mm, rotated rx 0 ry 90 rz 0 deg; joints [-12.688, -27.852, 110.223, -16.76, -81.829, 51.422]
  MoveL 8656 to (490.4, 509.6, 17) mm, rotated rx 0 ry 90 rz 0 deg; joints [-13.088, -28.22, 112.513, -17.092, -83.682, 50.903]
  Set speed (120.0 mm/s)
  MoveL 8657 to (490.4, 509.2, 17) mm, rotated rx 0 ry 90 rz 0 deg; joints [-13.051, -28.222, 112.524, -17.055, -83.689, 50.897]
  Set speed (1000.0 mm/s)
  MoveL 8658 to (491.1, 508.9, 17) mm, rotated rx 0 ry 90 rz 0 deg; joints [-13.008, -28.211, 112.45, -17.014, -83.627, 50.911]
  Set speed (1000.0 mm/s)
  MoveL 8659 to (490.68, 490.68, 17) mm, rotated rx 0 ry 90 rz 0 deg; joints [-11.324, -28.286, 112.964, -15.307, -84.004, 50.631]
  Set speed (1000.0 mm/s)
  MoveL 8660 to (490.68, 490.68, 17.1) mm, rotated rx 0 ry 90 rz 0 deg; joints [-11.324, -28.297, 112.97, -15.307, -83.999, 50.633]
  Set speed (30.0 mm/s)
  Call Extruder(0.767)
  MoveL 8661 to (509.32, 509.32, 17.1) mm, rotated rx 0 ry 90 rz 0 deg; joints [-12.669, -27.87, 110.27, -16.739, -81.856, 51.411]
  MoveL 8662 to (509.44, 509.44, 17.1) mm, rotated rx 0 ry 90 rz 0 deg; joints [-12.677, -27.867, 110.251, -16.749, -81.842, 51.417]
  Set speed (120.0 mm/s)
  MoveL 8663 to (509.32, 500.58, 17.1) mm, rotated rx 0 ry 90 rz 0 deg; joints [-11.882, -27.909, 110.499, -15.938, -82.009, 51.258]
  Set speed (30.0 mm/s)
  Call Extruder(0.360)
  MoveL 8664 to (500.58, 509.32, 17.1) mm, rotated rx 0 ry 90 rz 0 deg; joints [-12.847, -28.045, 111.318, -16.885, -82.698, 51.178]
  Set speed (120.0 mm/s)
  MoveL 8665 to (499.42, 509.32, 17.1) mm, rotated rx 0 ry 90 rz 0 deg; joints [-12.872, -28.067, 111.456, -16.905, -82.81, 51.147]
  Set speed (30.0 mm/s)
  Call Extruder(0.360)
  MoveL 8666 to (490.68, 500.58, 17.1) mm, rotated rx 0 ry 90 rz 0 deg; joints [-12.247, -28.261, 112.725, -16.241, -83.821, 50.774]
  Set speed (120.0 mm/s)
  MoveL 8667 to (490.68, 499.42, 17.1) mm, rotated rx 0 ry 90 rz 0 deg; joints [-12.139, -28.265, 112.755, -16.132, -83.843, 50.757]
  Set speed (30.0 mm/s)
  MoveL 8668 to (499.42, 490.68, 17.1) mm, rotated rx 0 ry 90 rz 0 deg; joints [-11.163, -28.141, 111.93, -15.171, -83.141, 50.851]
  Set speed (120.0 mm/s)
  MoveL 8669 to (500.58, 490.68, 17.1) mm, rotated rx 0 ry 90 rz 0 deg; joints [-11.141, -28.12, 111.791, -15.153, -83.027, 50.879]
  Set speed (30.0 mm/s)
  Call Extruder(0.360)
  MoveL 8670 to (509.32, 499.42, 17.1) mm, rotated rx 0 ry 90 rz 0 deg; joints [-11.777, -27.914, 110.528, -15.831, -82.029, 51.238]
  MoveL 8671 to (509.44, 499.54, 17.1) mm, rotated rx 0 ry 90 rz 0 deg; joints [-11.786, -27.911, 110.51, -15.841, -82.015, 51.243]
  Set speed (120.0 mm/s)
  MoveL 8672 to (509.32, 490.68, 17.1) mm, rotated rx 0 ry 90 rz 0 deg; joints [-10.985, -27.95, 110.741, -15.026, -82.172, 51.093]
  Set speed (30.0 mm/s)
  Call Extruder(0.767)
  MoveL 8673 to (490.68, 509.32, 17.1) mm, rotated rx 0 ry 90 rz 0 deg; joints [-13.056, -28.227, 112.493, -17.061, -83.655, 50.908]
  MoveL 8674 to (490.56, 509.44, 17.1) mm, rotated rx 0 ry 90 rz 0 deg; joints [-13.07, -28.229, 112.504, -17.074, -83.664, 50.906]
  Set speed (120.0 mm/s)
  MoveL 8675 to (490.4, 509.6, 17.1) mm, rotated rx 0 ry 90 rz 0 deg; joints [-13.088, -28.231, 112.518, -17.092, -83.676, 50.905]
  Set speed (15.0 mm/s)
  Call Extruder(0.559)
  MoveL 8676 to (490.4, 490.4, 17.1) mm, rotated rx 0 ry 90 rz 0 deg; joints [-11.303, -28.302, 113.009, -15.285, -84.031, 50.622]
  MoveL 8677 to (509.6, 490.4, 17.1) mm, rotated rx 0 ry 90 rz 0 deg; joints [-10.955, -27.945, 110.713, -14.996, -82.149, 51.095]
  MoveL 8678 to (509.6, 509.6, 17.1) mm, rotated rx 0 ry 90 rz 0 deg; joints [-12.688, -27.863, 110.228, -16.761, -81.824, 51.424]
  MoveL 8679 to (490.4, 509.6, 17.1) mm, rotated rx 0 ry 90 rz 0 deg; joints [-13.088, -28.231, 112.518, -17.092, -83.676, 50.905]
  Set speed (120.0 mm/s)
  MoveL 8680 to (490.4, 509.2, 17.1) mm, rotated rx 0 ry 90 rz 0 deg; joints [-13.051, -28.232, 112.529, -17.055, -83.684, 50.898]
  Set speed (1000.0 mm/s)
  MoveL 8681 to (491.1, 508.9, 17.1) mm, rotated rx 0 ry 90 rz 0 deg; joints [-13.008, -28.221, 112.455, -17.014, -83.622, 50.913]
  Set speed (1000.0 mm/s)
  MoveL 8682 to (490.68, 490.68, 17.1) mm, rotated rx 0 ry 90 rz 0 deg; joints [-11.324, -28.297, 112.97, -15.307, -83.999, 50.633]
  Set speed (1000.0 mm/s)
  MoveL 8683 to (490.68, 490.68, 17.2) mm, rotated rx 0 ry 90 rz 0 deg; joints [-11.324, -28.307, 112.975, -15.307, -83.993, 50.634]
  Set speed (30.0 mm/s)
  Call Extruder(0.767)
  MoveL 8684 to (509.32, 509.32, 17.2) mm, rotated rx 0 ry 90 rz 0 deg; joints [-12.669, -27.88, 110.275, -16.74, -81.85, 51.413]
  MoveL 8685 to (509.44, 509.44, 17.2) mm, rotated rx 0 ry 90 rz 0 deg; joints [-12.677, -27.877, 110.256, -16.749, -81.836, 51.418]
  Set speed (120.0 mm/s)
  MoveL 8686 to (509.32, 500.58, 17.2) mm, rotated rx 0 ry 90 rz 0 deg; joints [-11.882, -27.919, 110.504, -15.938, -82.004, 51.259]
  Set speed (30.0 mm/s)
  Call Extruder(0.360)
  MoveL 8687 to (500.58, 509.32, 17.2) mm, rotated rx 0 ry 90 rz 0 deg; joints [-12.847, -28.055, 111.323, -16.886, -82.693, 51.18]
  Set speed (120.0 mm/s)
  MoveL 8688 to (499.42, 509.32, 17.2) mm, rotated rx 0 ry 90 rz 0 deg; joints [-12.872, -28.077, 111.461, -16.906, -82.805, 51.148]
  Set speed (30.0 mm/s)
  Call Extruder(0.360)
  MoveL 8689 to (490.68, 500.58, 17.2) mm, rotated rx 0 ry 90 rz 0 deg; joints [-12.247, -28.272, 112.73, -16.241, -83.816, 50.776]
  Set speed (120.0 mm/s)
  MoveL 8690 to (490.68, 499.42, 17.2) mm, rotated rx 0 ry 90 rz 0 deg; joints [-12.139, -28.276, 112.76, -16.132, -83.837, 50.759]
  Set speed (30.0 mm/s)
  MoveL 8691 to (499.42, 490.68, 17.2) mm, rotated rx 0 ry 90 rz 0 deg; joints [-11.163, -28.152, 111.935, -15.171, -83.136, 50.852]
  Set speed (120.0 mm/s)
  MoveL 8692 to (500.58, 490.68, 17.2) mm, rotated rx 0 ry 90 rz 0 deg; joints [-11.141, -28.13, 111.796, -15.154, -83.022, 50.881]
  Set speed (30.0 mm/s)
  Call Extruder(0.360)
  MoveL 8693 to (509.32, 499.42, 17.2) mm, rotated rx 0 ry 90 rz 0 deg; joints [-11.777, -27.924, 110.533, -15.831, -82.024, 51.239]
  MoveL 8694 to (509.44, 499.54, 17.2) mm, rotated rx 0 ry 90 rz 0 deg; joints [-11.786, -27.921, 110.515, -15.841, -82.01, 51.245]
  Set speed (120.0 mm/s)
  MoveL 8695 to (509.32, 490.68, 17.2) mm, rotated rx 0 ry 90 rz 0 deg; joints [-10.985, -27.96, 110.746, -15.026, -82.167, 51.094]
  Set speed (30.0 mm/s)
  Call Extruder(0.767)
  MoveL 8696 to (490.68, 509.32, 17.2) mm, rotated rx 0 ry 90 rz 0 deg; joints [-13.056, -28.238, 112.498, -17.061, -83.649, 50.909]
  MoveL 8697 to (490.56, 509.44, 17.2) mm, rotated rx 0 ry 90 rz 0 deg; joints [-13.07, -28.239, 112.51, -17.075, -83.659, 50.908]
  Set speed (120.0 mm/s)
  MoveL 8698 to (490.4, 509.6, 17.2) mm, rotated rx 0 ry 90 rz 0 deg; joints [-13.088, -28.241, 112.524, -17.092, -83.671, 50.906]
  Set speed (15.0 mm/s)
  Call Extruder(0.559)
  MoveL 8699 to (490.4, 490.4, 17.2) mm, rotated rx 0 ry 90 rz 0 deg; joints [-11.303, -28.313, 113.014, -15.285, -84.026, 50.623]
  MoveL 8700 to (509.6, 490.4, 17.2) mm, rotated rx 0 ry 90 rz 0 deg; joints [-10.955, -27.956, 110.718, -14.996, -82.144, 51.096]
  MoveL 8701 to (509.6, 509.6, 17.2) mm, rotated rx 0 ry 90 rz 0 deg; joints [-12.688, -27.873, 110.233, -16.761, -81.818, 51.425]
  MoveL 8702 to (490.4, 509.6, 17.2) mm, rotated rx 0 ry 90 rz 0 deg; joints [-13.088, -28.241, 112.524, -17.092, -83.671, 50.906]
  Set speed (120.0 mm/s)
  MoveL 8703 to (490.4, 509.2, 17.2) mm, rotated rx 0 ry 90 rz 0 deg; joints [-13.051, -28.243, 112.535, -17.055, -83.679, 50.9]
  Set speed (1000.0 mm/s)
  MoveL 8704 to (491.1, 508.9, 17.2) mm, rotated rx 0 ry 90 rz 0 deg; joints [-13.008, -28.232, 112.46, -17.014, -83.617, 50.914]
  Set speed (1000.0 mm/s)
  MoveL 8705 to (490.68, 490.68, 17.2) mm, rotated rx 0 ry 90 rz 0 deg; joints [-11.324, -28.307, 112.975, -15.307, -83.993, 50.634]
  Set speed (1000.0 mm/s)
  MoveL 8706 to (490.68, 490.68, 17.3) mm, rotated rx 0 ry 90 rz 0 deg; joints [-11.324, -28.318, 112.98, -15.307, -83.988, 50.636]
  Set speed (30.0 mm/s)
  Call Extruder(0.287)
  MoveL 8707 to (497.65, 497.65, 17.3) mm, rotated rx 0 ry 90 rz 0 deg; joints [-11.838, -28.169, 111.981, -15.851, -83.184, 50.915]
  MoveL 8708 to (497.78, 497.78, 17.3) mm, rotated rx 0 ry 90 rz 0 deg; joints [-11.847, -28.166, 111.964, -15.86, -83.17, 50.92]
  Set speed (120.0 mm/s)
  MoveL 8709 to (499.24, 500.76, 17.3) mm, rotated rx 0 ry 90 rz 0 deg; joints [-12.093, -28.127, 111.714, -16.115, -82.974, 51.005]
  Set speed (30.0 mm/s)
  Call Extruder(0.352)
  MoveL 8710 to (490.68, 509.32, 17.3) mm, rotated rx 0 ry 90 rz 0 deg; joints [-13.056, -28.248, 112.503, -17.061, -83.644, 50.911]
  MoveL 8711 to (490.56, 509.44, 17.3) mm, rotated rx 0 ry 90 rz 0 deg; joints [-13.07, -28.25, 112.515, -17.075, -83.654, 50.91]
  Set speed (120.0 mm/s)
  MoveL 8712 to (496.13, 506.03, 17.3) mm, rotated rx 0 ry 90 rz 0 deg; joints [-12.639, -28.164, 111.947, -16.657, -83.18, 51.007]
  Set speed (30.0 mm/s)
  Call Extruder(0.224)
  MoveL 8713 to (490.68, 500.58, 17.3) mm, rotated rx 0 ry 90 rz 0 deg; joints [-12.247, -28.282, 112.735, -16.241, -83.811, 50.777]
  Set speed (120.0 mm/s)
  MoveL 8714 to (490.68, 499.42, 17.3) mm, rotated rx 0 ry 90 rz 0 deg; joints [-12.139, -28.287, 112.765, -16.132, -83.832, 50.76]
  Set speed (30.0 mm/s)
  Call Extruder(0.215)
  MoveL 8715 to (495.89, 494.21, 17.3) mm, rotated rx 0 ry 90 rz 0 deg; joints [-11.554, -28.214, 112.276, -15.556, -83.416, 50.818]
  Set speed (120.0 mm/s)
  MoveL 8716 to (496.37, 493.73, 17.3) mm, rotated rx 0 ry 90 rz 0 deg; joints [-11.5, -28.207, 112.231, -15.504, -83.377, 50.823]
  Set speed (30.0 mm/s)
  Call Extruder(0.125)
  MoveL 8717 to (499.42, 490.68, 17.3) mm, rotated rx 0 ry 90 rz 0 deg; joints [-11.163, -28.163, 111.94, -15.171, -83.13, 50.854]
  Set speed (120.0 mm/s)
  MoveL 8718 to (500.58, 490.68, 17.3) mm, rotated rx 0 ry 90 rz 0 deg; joints [-11.141, -28.141, 111.801, -15.154, -83.017, 50.882]
  Set speed (30.0 mm/s)
  MoveL 8719 to (503.63, 493.73, 17.3) mm, rotated rx 0 ry 90 rz 0 deg; joints [-11.366, -28.071, 111.364, -15.392, -82.668, 51.005]
  Set speed (120.0 mm/s)
  MoveL 8720 to (504.39, 494.49, 17.3) mm, rotated rx 0 ry 90 rz 0 deg; joints [-11.421, -28.054, 111.253, -15.451, -82.581, 51.036]
  Set speed (30.0 mm/s)
  Call Extruder(0.203)
  MoveL 8721 to (509.32, 499.42, 17.3) mm, rotated rx 0 ry 90 rz 0 deg; joints [-11.777, -27.935, 110.538, -15.832, -82.018, 51.241]
  Set speed (120.0 mm/s)
  MoveL 8722 to (509.32, 500.58, 17.3) mm, rotated rx 0 ry 90 rz 0 deg; joints [-11.882, -27.93, 110.509, -15.938, -81.999, 51.261]
  Set speed (30.0 mm/s)
  Call Extruder(0.212)
  MoveL 8723 to (504.16, 505.74, 17.3) mm, rotated rx 0 ry 90 rz 0 deg; joints [-12.449, -28.011, 110.996, -16.495, -82.408, 51.216]
  Set speed (120.0 mm/s)
  MoveL 8724 to (503.3, 506.6, 17.3) mm, rotated rx 0 ry 90 rz 0 deg; joints [-12.544, -28.025, 111.076, -16.588, -82.475, 51.208]
  Set speed (30.0 mm/s)
  Call Extruder(0.112)
  MoveL 8725 to (500.58, 509.32, 17.3) mm, rotated rx 0 ry 90 rz 0 deg; joints [-12.847, -28.066, 111.328, -16.886, -82.688, 51.181]
  Set speed (120.0 mm/s)
  MoveL 8726 to (499.42, 509.32, 17.3) mm, rotated rx 0 ry 90 rz 0 deg; joints [-12.872, -28.088, 111.466, -16.906, -82.8, 51.15]
  Set speed (30.0 mm/s)
  Call Extruder(0.112)
  MoveL 8727 to (496.7, 506.6, 17.3) mm, rotated rx 0 ry 90 rz 0 deg; joints [-12.679, -28.151, 111.864, -16.7, -83.114, 51.031]
  MoveL 8728 to (496.57, 506.47, 17.3) mm, rotated rx 0 ry 90 rz 0 deg; joints [-12.67, -28.153, 111.882, -16.691, -83.128, 51.026]
  Set speed (120.0 mm/s)
  MoveL 8729 to (502.51, 502.51, 17.3) mm, rotated rx 0 ry 90 rz 0 deg; joints [-12.188, -28.058, 111.278, -16.223, -82.626, 51.118]
  Set speed (30.0 mm/s)
  Call Extruder(0.280)
  MoveL 8730 to (509.32, 509.32, 17.3) mm, rotated rx 0 ry 90 rz 0 deg; joints [-12.669, -27.891, 110.28, -16.74, -81.845, 51.415]
  MoveL 8731 to (509.44, 509.44, 17.3) mm, rotated rx 0 ry 90 rz 0 deg; joints [-12.677, -27.888, 110.261, -16.749, -81.831, 51.42]
  Set speed (120.0 mm/s)
  MoveL 8732 to (500.81, 499.19, 17.3) mm, rotated rx 0 ry 90 rz 0 deg; joints [-11.919, -28.104, 111.566, -15.943, -82.849, 51.02]
  Set speed (30.0 mm/s)
  Call Extruder(0.140)
  MoveL 8733 to (504.2, 495.8, 17.3) mm, rotated rx 0 ry 90 rz 0 deg; joints [-11.544, -28.052, 111.245, -15.575, -82.578, 51.052]
  Set speed (120.0 mm/s)
  MoveL 8734 to (504.39, 495.61, 17.3) mm, rotated rx 0 ry 90 rz 0 deg; joints [-11.523, -28.049, 111.226, -15.555, -82.562, 51.054]
  Set speed (30.0 mm/s)
  Call Extruder(0.203)
  MoveL 8735 to (509.32, 490.68, 17.3) mm, rotated rx 0 ry 90 rz 0 deg; joints [-10.985, -27.971, 110.751, -15.026, -82.162, 51.095]
  MoveL 8736 to (509.44, 490.56, 17.3) mm, rotated rx 0 ry 90 rz 0 deg; joints [-10.972, -27.969, 110.739, -15.013, -82.152, 51.096]
  Set speed (120.0 mm/s)
  MoveL 8737 to (490.47, 509.53, 17.3) mm, rotated rx 0 ry 90 rz 0 deg; joints [-13.08, -28.251, 112.522, -17.085, -83.66, 50.909]
  Set speed (1000.0 mm/s)
  MoveL 8738 to (490.4, 509.6, 17.3) mm, rotated rx 0 ry 90 rz 0 deg; joints [-13.088, -28.252, 112.529, -17.092, -83.666, 50.908]
  Set speed (15.0 mm/s)
  Call Extruder(0.559)
  MoveL 8739 to (490.4, 490.4, 17.3) mm, rotated rx 0 ry 90 rz 0 deg; joints [-11.303, -28.324, 113.019, -15.285, -84.02, 50.625]
  MoveL 8740 to (509.6, 490.4, 17.3) mm, rotated rx 0 ry 90 rz 0 deg; joints [-10.955, -27.966, 110.723, -14.996, -82.139, 51.098]
  MoveL 8741 to (509.6, 509.6, 17.3) mm, rotated rx 0 ry 90 rz 0 deg; joints [-12.688, -27.884, 110.238, -16.761, -81.813, 51.427]
  MoveL 8742 to (490.4, 509.6, 17.3) mm, rotated rx 0 ry 90 rz 0 deg; joints [-13.088, -28.252, 112.529, -17.092, -83.666, 50.908]
  Set speed (120.0 mm/s)
  MoveL 8743 to (490.4, 509.2, 17.3) mm, rotated rx 0 ry 90 rz 0 deg; joints [-13.051, -28.254, 112.54, -17.055, -83.673, 50.901]
  Set speed (1000.0 mm/s)
  MoveL 8744 to (490.5, 509.2, 17.3) mm, rotated rx 0 ry 90 rz 0 deg; joints [-13.049, -28.252, 112.528, -17.053, -83.664, 50.904]
  Set speed (1000.0 mm/s)
  MoveL 8745 to (496.05, 506.68, 17.3) mm, rotated rx 0 ry 90 rz 0 deg; joints [-12.7, -28.162, 111.939, -16.719, -83.176, 51.015]
  Set speed (15.0 mm/s)
  Call Extruder(0.065)
  MoveL 8746 to (496.05, 504.44, 17.3) mm, rotated rx 0 ry 90 rz 0 deg; joints [-12.495, -28.172, 111.998, -16.511, -83.217, 50.979]
  Call Extruder(0.145)
  MoveL 8747 to (501.03, 504.44, 17.3) mm, rotated rx 0 ry 90 rz 0 deg; joints [-12.394, -28.078, 111.405, -16.427, -82.734, 51.111]
  Call Extruder(0.353)
  MoveL 8748 to (495.52, 493.65, 17.3) mm, rotated rx 0 ry 90 rz 0 deg; joints [-11.509, -28.223, 112.334, -15.51, -83.462, 50.8]
  Call Extruder(0.261)
  MoveL 8749 to (504.47, 493.65, 17.3) mm, rotated rx 0 ry 90 rz 0 deg; joints [-11.343, -28.055, 111.264, -15.372, -82.587, 51.025]
  Call Extruder(0.065)
  MoveL 8750 to (504.47, 495.88, 17.3) mm, rotated rx 0 ry 90 rz 0 deg; joints [-11.547, -28.046, 111.21, -15.579, -82.55, 51.06]
  Call Extruder(0.153)
  MoveL 8751 to (499.21, 495.88, 17.3) mm, rotated rx 0 ry 90 rz 0 deg; joints [-11.646, -28.147, 111.84, -15.66, -83.063, 50.927]
  Call Extruder(0.353)
  MoveL 8752 to (504.73, 506.68, 17.3) mm, rotated rx 0 ry 90 rz 0 deg; joints [-12.523, -27.996, 110.902, -16.572, -82.336, 51.247]
  Call Extruder(0.253)
  MoveL 8753 to (496.05, 506.68, 17.3) mm, rotated rx 0 ry 90 rz 0 deg; joints [-12.7, -28.162, 111.939, -16.719, -83.176, 51.015]
  Set speed (120.0 mm/s)
  MoveL 8754 to (496.46, 506.36, 17.3) mm, rotated rx 0 ry 90 rz 0 deg; joints [-12.662, -28.156, 111.898, -16.682, -83.141, 51.021]
  Set speed (15.0 mm/s)
  Call Extruder(0.004)
  MoveL 8755 to (496.36, 506.26, 17.3) mm, rotated rx 0 ry 90 rz 0 deg; joints [-12.655, -28.158, 111.913, -16.675, -83.153, 51.017]
  Set speed (120.0 mm/s)
  MoveL 8756 to (496.36, 505.27, 17.3) mm, rotated rx 0 ry 90 rz 0 deg; joints [-12.564, -28.162, 111.939, -16.583, -83.171, 51.001]
  Set speed (15.0 mm/s)
  Call Extruder(0.045)
  MoveL 8757 to (497.45, 506.36, 17.3) mm, rotated rx 0 ry 90 rz 0 deg; joints [-12.642, -28.138, 111.78, -16.665, -83.045, 51.048]
  Set speed (120.0 mm/s)
  MoveL 8758 to (498.44, 506.36, 17.3) mm, rotated rx 0 ry 90 rz 0 deg; joints [-12.622, -28.119, 111.663, -16.648, -82.95, 51.074]
  Set speed (15.0 mm/s)
  Call Extruder(0.066)
  MoveL 8759 to (496.84, 504.76, 17.3) mm, rotated rx 0 ry 90 rz 0 deg; joints [-12.508, -28.156, 111.896, -16.527, -83.135, 51.006]
  Set speed (120.0 mm/s)
  MoveL 8760 to (497.83, 504.76, 17.3) mm, rotated rx 0 ry 90 rz 0 deg; joints [-12.488, -28.137, 111.778, -16.51, -83.039, 51.032]
  Set speed (15.0 mm/s)
  MoveL 8761 to (499.43, 506.36, 17.3) mm, rotated rx 0 ry 90 rz 0 deg; joints [-12.602, -28.1, 111.545, -16.632, -82.854, 51.101]
  Set speed (120.0 mm/s)
  MoveL 8762 to (500.42, 506.36, 17.3) mm, rotated rx 0 ry 90 rz 0 deg; joints [-12.581, -28.081, 111.426, -16.615, -82.758, 51.127]
  Set speed (15.0 mm/s)
  MoveL 8763 to (498.82, 504.76, 17.3) mm, rotated rx 0 ry 90 rz 0 deg; joints [-12.468, -28.119, 111.66, -16.493, -82.943, 51.058]
  Set speed (120.0 mm/s)
  MoveL 8764 to (499.81, 504.76, 17.3) mm, rotated rx 0 ry 90 rz 0 deg; joints [-12.448, -28.1, 111.542, -16.476, -82.847, 51.084]
  Set speed (15.0 mm/s)
  MoveL 8765 to (501.41, 506.36, 17.3) mm, rotated rx 0 ry 90 rz 0 deg; joints [-12.561, -28.062, 111.308, -16.598, -82.662, 51.154]
  Set speed (120.0 mm/s)
  MoveL 8766 to (502.4, 506.36, 17.3) mm, rotated rx 0 ry 90 rz 0 deg; joints [-12.541, -28.043, 111.19, -16.582, -82.566, 51.18]
  Set speed (15.0 mm/s)
  MoveL 8767 to (500.8, 504.76, 17.3) mm, rotated rx 0 ry 90 rz 0 deg; joints [-12.428, -28.081, 111.424, -16.46, -82.751, 51.111]
  Set speed (120.0 mm/s)
  MoveL 8768 to (501.28, 504.25, 17.3) mm, rotated rx 0 ry 90 rz 0 deg; joints [-12.372, -28.074, 111.379, -16.405, -82.713, 51.115]
  Set speed (15.0 mm/s)
  Call Extruder(0.087)
  MoveL 8769 to (503.39, 506.36, 17.3) mm, rotated rx 0 ry 90 rz 0 deg; joints [-12.521, -28.024, 111.071, -16.565, -82.471, 51.206]
  Set speed (120.0 mm/s)
  MoveL 8770 to (504.04, 506.02, 17.3) mm, rotated rx 0 ry 90 rz 0 deg; joints [-12.477, -28.013, 111.003, -16.523, -82.414, 51.217]
  Set speed (15.0 mm/s)
  Call Extruder(0.156)
  MoveL 8771 to (500.25, 502.23, 17.3) mm, rotated rx 0 ry 90 rz 0 deg; joints [-12.208, -28.102, 111.555, -16.235, -82.85, 51.055]
  MoveL 8772 to (500.13, 502.11, 17.3) mm, rotated rx 0 ry 90 rz 0 deg; joints [-12.199, -28.105, 111.573, -16.225, -82.864, 51.05]
  Set speed (120.0 mm/s)
  MoveL 8773 to (501.96, 501.96, 17.3) mm, rotated rx 0 ry 90 rz 0 deg; joints [-12.15, -28.07, 111.357, -16.182, -82.688, 51.095]
  Set speed (15.0 mm/s)
  Call Extruder(0.155)
  MoveL 8774 to (498.19, 498.19, 17.3) mm, rotated rx 0 ry 90 rz 0 deg; joints [-11.878, -28.157, 111.904, -15.892, -83.122, 50.937]
  MoveL 8775 to (498.07, 498.07, 17.3) mm, rotated rx 0 ry 90 rz 0 deg; joints [-11.869, -28.16, 111.922, -15.883, -83.136, 50.932]
  Set speed (120.0 mm/s)
  MoveL 8776 to (499.89, 497.91, 17.3) mm, rotated rx 0 ry 90 rz 0 deg; joints [-11.819, -28.126, 111.708, -15.839, -82.961, 50.976]
  Set speed (15.0 mm/s)
  Call Extruder(0.155)
  MoveL 8777 to (496.13, 494.15, 17.3) mm, rotated rx 0 ry 90 rz 0 deg; joints [-11.544, -28.21, 112.249, -15.547, -83.394, 50.823]
  Set speed (120.0 mm/s)
  MoveL 8778 to (496.93, 493.96, 17.3) mm, rotated rx 0 ry 90 rz 0 deg; joints [-11.512, -28.196, 112.158, -15.517, -83.318, 50.841]
  Set speed (15.0 mm/s)
  Call Extruder(0.079)
  MoveL 8779 to (498.85, 495.88, 17.3) mm, rotated rx 0 ry 90 rz 0 deg; joints [-11.652, -28.154, 111.883, -15.666, -83.098, 50.918]
  Set speed (120.0 mm/s)
  MoveL 8780 to (499.52, 495.57, 17.3) mm, rotated rx 0 ry 90 rz 0 deg; joints [-11.611, -28.142, 111.81, -15.626, -83.038, 50.931]
  Set speed (15.0 mm/s)
  Call Extruder(0.066)
  MoveL 8781 to (497.92, 493.96, 17.3) mm, rotated rx 0 ry 90 rz 0 deg; joints [-11.493, -28.178, 112.04, -15.501, -83.222, 50.866]
  Set speed (120.0 mm/s)
  MoveL 8782 to (498.91, 493.96, 17.3) mm, rotated rx 0 ry 90 rz 0 deg; joints [-11.475, -28.16, 111.922, -15.486, -83.125, 50.891]
  Set speed (15.0 mm/s)
  MoveL 8783 to (500.51, 495.57, 17.3) mm, rotated rx 0 ry 90 rz 0 deg; joints [-11.592, -28.124, 111.692, -15.61, -82.941, 50.956]
  Set speed (120.0 mm/s)
  MoveL 8784 to (501.5, 495.57, 17.3) mm, rotated rx 0 ry 90 rz 0 deg; joints [-11.573, -28.105, 111.573, -15.595, -82.844, 50.981]
  Set speed (15.0 mm/s)
  MoveL 8785 to (499.9, 493.96, 17.3) mm, rotated rx 0 ry 90 rz 0 deg; joints [-11.456, -28.141, 111.804, -15.471, -83.028, 50.915]
  Set speed (120.0 mm/s)
  MoveL 8786 to (500.89, 493.96, 17.3) mm, rotated rx 0 ry 90 rz 0 deg; joints [-11.438, -28.123, 111.686, -15.455, -82.931, 50.94]
  Set speed (15.0 mm/s)
  MoveL 8787 to (502.49, 495.57, 17.3) mm, rotated rx 0 ry 90 rz 0 deg; joints [-11.555, -28.086, 111.455, -15.58, -82.748, 51.006]
  Set speed (120.0 mm/s)
  MoveL 8788 to (503.48, 495.56, 17.3) mm, rotated rx 0 ry 90 rz 0 deg; joints [-11.536, -28.067, 111.336, -15.565, -82.651, 51.03]
  Set speed (15.0 mm/s)
  MoveL 8789 to (501.88, 493.96, 17.3) mm, rotated rx 0 ry 90 rz 0 deg; joints [-11.419, -28.104, 111.567, -15.44, -82.835, 50.965]
  Set speed (120.0 mm/s)
  MoveL 8790 to (502.87, 493.96, 17.3) mm, rotated rx 0 ry 90 rz 0 deg; joints [-11.401, -28.085, 111.448, -15.425, -82.738, 50.99]
  Set speed (15.0 mm/s)
  Call Extruder(0.053)
  MoveL 8791 to (504.16, 495.25, 17.3) mm, rotated rx 0 ry 90 rz 0 deg; joints [-11.495, -28.055, 111.263, -15.525, -82.591, 51.042]
  Set speed (120.0 mm/s)
  MoveL 8792 to (504.16, 494.26, 17.3) mm, rotated rx 0 ry 90 rz 0 deg; joints [-11.404, -28.059, 111.287, -15.433, -82.608, 51.026]
  Set speed (15.0 mm/s)
  Call Extruder(0.012)
  MoveL 8793 to (503.86, 493.96, 17.3) mm, rotated rx 0 ry 90 rz 0 deg; joints [-11.383, -28.066, 111.33, -15.41, -82.641, 51.014]
  Set speed (120.0 mm/s)
  MoveL 8794 to (500.93, 499.94, 17.3) mm, rotated rx 0 ry 90 rz 0 deg; joints [-11.985, -28.099, 111.533, -16.011, -82.825, 51.035]
  Set speed (15.0 mm/s)
  Call Extruder(0.155)
  MoveL 8795 to (497.16, 496.17, 17.3) mm, rotated rx 0 ry 90 rz 0 deg; joints [-11.711, -28.184, 112.077, -15.72, -83.258, 50.88]
  MoveL 8796 to (497.04, 496.05, 17.3) mm, rotated rx 0 ry 90 rz 0 deg; joints [-11.702, -28.186, 112.095, -15.71, -83.272, 50.875]
  Set speed (120.0 mm/s)
  MoveL 8797 to (499.22, 500.21, 17.3) mm, rotated rx 0 ry 90 rz 0 deg; joints [-12.043, -28.13, 111.73, -16.064, -82.986, 50.996]
  Set speed (15.0 mm/s)
  Call Extruder(0.156)
  MoveL 8798 to (503, 503.99, 17.3) mm, rotated rx 0 ry 90 rz 0 deg; joints [-12.314, -28.042, 111.18, -16.353, -82.551, 51.156]
  MoveL 8799 to (503.12, 504.12, 17.3) mm, rotated rx 0 ry 90 rz 0 deg; joints [-12.323, -28.039, 111.162, -16.362, -82.537, 51.161]
  Set speed (120.0 mm/s)
  MoveL 8800 to (490.68, 490.68, 17.3) mm, rotated rx 0 ry 90 rz 0 deg; joints [-11.324, -28.318, 112.98, -15.307, -83.988, 50.636]
  Set speed (1000.0 mm/s)
  MoveL 8801 to (490.68, 490.68, 17.4) mm, rotated rx 0 ry 90 rz 0 deg; joints [-11.324, -28.329, 112.985, -15.308, -83.983, 50.637]
  Set speed (30.0 mm/s)
  Call Extruder(0.287)
  MoveL 8802 to (497.65, 497.65, 17.4) mm, rotated rx 0 ry 90 rz 0 deg; joints [-11.838, -28.18, 111.987, -15.851, -83.178, 50.917]
  MoveL 8803 to (497.78, 497.78, 17.4) mm, rotated rx 0 ry 90 rz 0 deg; joints [-11.847, -28.177, 111.969, -15.86, -83.164, 50.922]
  Set speed (120.0 mm/s)
  MoveL 8804 to (499.24, 500.76, 17.4) mm, rotated rx 0 ry 90 rz 0 deg; joints [-12.093, -28.138, 111.719, -16.115, -82.969, 51.006]
  Set speed (30.0 mm/s)
  Call Extruder(0.352)
  MoveL 8805 to (490.68, 509.32, 17.4) mm, rotated rx 0 ry 90 rz 0 deg; joints [-13.056, -28.259, 112.509, -17.061, -83.639, 50.913]
  MoveL 8806 to (490.56, 509.44, 17.4) mm, rotated rx 0 ry 90 rz 0 deg; joints [-13.07, -28.261, 112.52, -17.075, -83.648, 50.911]
  Set speed (120.0 mm/s)
  MoveL 8807 to (496.13, 506.03, 17.4) mm, rotated rx 0 ry 90 rz 0 deg; joints [-12.639, -28.174, 111.952, -16.657, -83.175, 51.009]
  Set speed (30.0 mm/s)
  Call Extruder(0.224)
  MoveL 8808 to (490.68, 500.58, 17.4) mm, rotated rx 0 ry 90 rz 0 deg; joints [-12.247, -28.293, 112.74, -16.241, -83.805, 50.779]
  Set speed (120.0 mm/s)
  MoveL 8809 to (490.68, 499.42, 17.4) mm, rotated rx 0 ry 90 rz 0 deg; joints [-12.139, -28.297, 112.77, -16.132, -83.827, 50.762]
  Set speed (30.0 mm/s)
  Call Extruder(0.215)
  MoveL 8810 to (495.89, 494.2, 17.4) mm, rotated rx 0 ry 90 rz 0 deg; joints [-11.554, -28.225, 112.281, -15.556, -83.41, 50.819]
  Set speed (120.0 mm/s)
  MoveL 8811 to (496.37, 493.73, 17.4) mm, rotated rx 0 ry 90 rz 0 deg; joints [-11.5, -28.218, 112.236, -15.504, -83.372, 50.824]
  Set speed (30.0 mm/s)
  Call Extruder(0.125)
  MoveL 8812 to (499.42, 490.68, 17.4) mm, rotated rx 0 ry 90 rz 0 deg; joints [-11.163, -28.173, 111.945, -15.171, -83.125, 50.855]
  Set speed (120.0 mm/s)
  MoveL 8813 to (500.58, 490.68, 17.4) mm, rotated rx 0 ry 90 rz 0 deg; joints [-11.141, -28.151, 111.806, -15.154, -83.012, 50.884]
  Set speed (30.0 mm/s)
  MoveL 8814 to (503.63, 493.73, 17.4) mm, rotated rx 0 ry 90 rz 0 deg; joints [-11.366, -28.082, 111.369, -15.392, -82.663, 51.006]
  Set speed (120.0 mm/s)
  MoveL 8815 to (504.39, 494.49, 17.4) mm, rotated rx 0 ry 90 rz 0 deg; joints [-11.421, -28.064, 111.258, -15.451, -82.576, 51.037]
  Set speed (30.0 mm/s)
  Call Extruder(0.203)
  MoveL 8816 to (509.32, 499.42, 17.4) mm, rotated rx 0 ry 90 rz 0 deg; joints [-11.777, -27.945, 110.543, -15.832, -82.013, 51.242]
  Set speed (120.0 mm/s)
  MoveL 8817 to (509.32, 500.58, 17.4) mm, rotated rx 0 ry 90 rz 0 deg; joints [-11.882, -27.94, 110.514, -15.938, -81.994, 51.262]
  Set speed (30.0 mm/s)
  Call Extruder(0.212)
  MoveL 8818 to (504.16, 505.74, 17.4) mm, rotated rx 0 ry 90 rz 0 deg; joints [-12.449, -28.022, 111.001, -16.495, -82.403, 51.217]
  Set speed (120.0 mm/s)
  MoveL 8819 to (503.3, 506.6, 17.4) mm, rotated rx 0 ry 90 rz 0 deg; joints [-12.544, -28.035, 111.081, -16.589, -82.47, 51.209]
  Set speed (30.0 mm/s)
  Call Extruder(0.112)
  MoveL 8820 to (500.58, 509.32, 17.4) mm, rotated rx 0 ry 90 rz 0 deg; joints [-12.847, -28.076, 111.333, -16.886, -82.683, 51.183]
  Set speed (120.0 mm/s)
  MoveL 8821 to (499.42, 509.32, 17.4) mm, rotated rx 0 ry 90 rz 0 deg; joints [-12.872, -28.098, 111.471, -16.906, -82.795, 51.151]
  Set speed (30.0 mm/s)
  Call Extruder(0.112)
  MoveL 8822 to (496.7, 506.6, 17.4) mm, rotated rx 0 ry 90 rz 0 deg; joints [-12.679, -28.161, 111.869, -16.7, -83.109, 51.033]
  MoveL 8823 to (496.57, 506.47, 17.4) mm, rotated rx 0 ry 90 rz 0 deg; joints [-12.67, -28.164, 111.887, -16.691, -83.123, 51.028]
  Set speed (120.0 mm/s)
  MoveL 8824 to (502.51, 502.51, 17.4) mm, rotated rx 0 ry 90 rz 0 deg; joints [-12.188, -28.068, 111.283, -16.224, -82.621, 51.12]
  Set speed (30.0 mm/s)
  Call Extruder(0.280)
  MoveL 8825 to (509.32, 509.32, 17.4) mm, rotated rx 0 ry 90 rz 0 deg; joints [-12.669, -27.901, 110.285, -16.74, -81.84, 51.416]
  MoveL 8826 to (509.44, 509.44, 17.4) mm, rotated rx 0 ry 90 rz 0 deg; joints [-12.677, -27.898, 110.267, -16.749, -81.826, 51.422]
  Set speed (120.0 mm/s)
  MoveL 8827 to (500.81, 499.19, 17.4) mm, rotated rx 0 ry 90 rz 0 deg; joints [-11.919, -28.114, 111.571, -15.943, -82.844, 51.022]
  Set speed (30.0 mm/s)
  Call Extruder(0.140)
  MoveL 8828 to (504.2, 495.8, 17.4) mm, rotated rx 0 ry 90 rz 0 deg; joints [-11.544, -28.063, 111.25, -15.576, -82.572, 51.054]
  Set speed (120.0 mm/s)
  MoveL 8829 to (504.39, 495.61, 17.4) mm, rotated rx 0 ry 90 rz 0 deg; joints [-11.523, -28.06, 111.231, -15.555, -82.557, 51.055]
  Set speed (30.0 mm/s)
  Call Extruder(0.203)
  MoveL 8830 to (509.32, 490.68, 17.4) mm, rotated rx 0 ry 90 rz 0 deg; joints [-10.985, -27.981, 110.756, -15.026, -82.157, 51.097]
  MoveL 8831 to (509.44, 490.56, 17.4) mm, rotated rx 0 ry 90 rz 0 deg; joints [-10.972, -27.979, 110.744, -15.013, -82.147, 51.098]
  Set speed (120.0 mm/s)
  MoveL 8832 to (490.47, 509.53, 17.4) mm, rotated rx 0 ry 90 rz 0 deg; joints [-13.08, -28.262, 112.527, -17.085, -83.655, 50.91]
  Set speed (1000.0 mm/s)
  MoveL 8833 to (490.4, 509.6, 17.4) mm, rotated rx 0 ry 90 rz 0 deg; joints [-13.088, -28.263, 112.534, -17.093, -83.66, 50.909]
  Set speed (15.0 mm/s)
  Call Extruder(0.559)
  MoveL 8834 to (490.4, 490.4, 17.4) mm, rotated rx 0 ry 90 rz 0 deg; joints [-11.303, -28.334, 113.025, -15.286, -84.015, 50.626]
  MoveL 8835 to (509.6, 490.4, 17.4) mm, rotated rx 0 ry 90 rz 0 deg; joints [-10.955, -27.977, 110.728, -14.997, -82.134, 51.099]
  MoveL 8836 to (509.6, 509.6, 17.4) mm, rotated rx 0 ry 90 rz 0 deg; joints [-12.688, -27.894, 110.243, -16.761, -81.808, 51.429]
  MoveL 8837 to (490.4, 509.6, 17.4) mm, rotated rx 0 ry 90 rz 0 deg; joints [-13.088, -28.263, 112.534, -17.093, -83.66, 50.909]
  Set speed (120.0 mm/s)
  MoveL 8838 to (490.4, 509.2, 17.4) mm, rotated rx 0 ry 90 rz 0 deg; joints [-13.051, -28.264, 112.545, -17.055, -83.668, 50.903]
  Set speed (1000.0 mm/s)
  MoveL 8839 to (490.5, 509.2, 17.4) mm, rotated rx 0 ry 90 rz 0 deg; joints [-13.049, -28.262, 112.533, -17.053, -83.658, 50.906]
  Set speed (1000.0 mm/s)
  MoveL 8840 to (496.05, 506.68, 17.4) mm, rotated rx 0 ry 90 rz 0 deg; joints [-12.7, -28.173, 111.944, -16.719, -83.17, 51.017]
  Set speed (15.0 mm/s)
  Call Extruder(0.065)
  MoveL 8841 to (496.05, 504.44, 17.4) mm, rotated rx 0 ry 90 rz 0 deg; joints [-12.495, -28.182, 112.004, -16.511, -83.212, 50.981]
  Call Extruder(0.145)
  MoveL 8842 to (501.03, 504.45, 17.4) mm, rotated rx 0 ry 90 rz 0 deg; joints [-12.394, -28.089, 111.41, -16.427, -82.729, 51.113]
  Call Extruder(0.353)
  MoveL 8843 to (495.52, 493.65, 17.4) mm, rotated rx 0 ry 90 rz 0 deg; joints [-11.509, -28.233, 112.339, -15.51, -83.457, 50.802]
  Call Extruder(0.261)
  MoveL 8844 to (504.47, 493.65, 17.4) mm, rotated rx 0 ry 90 rz 0 deg; joints [-11.343, -28.066, 111.269, -15.372, -82.582, 51.026]
  Call Extruder(0.065)
  MoveL 8845 to (504.47, 495.88, 17.4) mm, rotated rx 0 ry 90 rz 0 deg; joints [-11.547, -28.057, 111.215, -15.579, -82.544, 51.062]
  Call Extruder(0.153)
  MoveL 8846 to (499.21, 495.88, 17.4) mm, rotated rx 0 ry 90 rz 0 deg; joints [-11.646, -28.158, 111.845, -15.661, -83.058, 50.929]
  Call Extruder(0.353)
  MoveL 8847 to (504.73, 506.68, 17.4) mm, rotated rx 0 ry 90 rz 0 deg; joints [-12.523, -28.006, 110.907, -16.573, -82.33, 51.248]
  Call Extruder(0.253)
  MoveL 8848 to (496.05, 506.68, 17.4) mm, rotated rx 0 ry 90 rz 0 deg; joints [-12.7, -28.173, 111.944, -16.719, -83.17, 51.017]
  Set speed (120.0 mm/s)
  MoveL 8849 to (503.93, 505.81, 17.4) mm, rotated rx 0 ry 90 rz 0 deg; joints [-12.461, -28.026, 111.026, -16.506, -82.423, 51.213]
  Set speed (15.0 mm/s)
  Call Extruder(0.023)
  MoveL 8850 to (503.39, 506.36, 17.4) mm, rotated rx 0 ry 90 rz 0 deg; joints [-12.521, -28.034, 111.077, -16.566, -82.466, 51.207]
  Set speed (120.0 mm/s)
  MoveL 8851 to (502.4, 506.36, 17.4) mm, rotated rx 0 ry 90 rz 0 deg; joints [-12.541, -28.054, 111.195, -16.582, -82.562, 51.181]
  Set speed (15.0 mm/s)
  Call Extruder(0.049)
  MoveL 8852 to (503.6, 505.16, 17.4) mm, rotated rx 0 ry 90 rz 0 deg; joints [-12.408, -28.035, 111.083, -16.451, -82.467, 51.193]
  Set speed (120.0 mm/s)
  MoveL 8853 to (503.26, 504.5, 17.4) mm, rotated rx 0 ry 90 rz 0 deg; joints [-12.355, -28.045, 111.141, -16.396, -82.511, 51.173]
  Set speed (15.0 mm/s)
  Call Extruder(0.076)
  MoveL 8854 to (501.41, 506.36, 17.4) mm, rotated rx 0 ry 90 rz 0 deg; joints [-12.561, -28.073, 111.314, -16.598, -82.658, 51.155]
  Set speed (120.0 mm/s)
  MoveL 8855 to (500.42, 506.36, 17.4) mm, rotated rx 0 ry 90 rz 0 deg; joints [-12.581, -28.092, 111.432, -16.615, -82.753, 51.129]
  Set speed (15.0 mm/s)
  Call Extruder(0.103)
  MoveL 8856 to (502.93, 503.85, 17.4) mm, rotated rx 0 ry 90 rz 0 deg; joints [-12.302, -28.054, 111.198, -16.341, -82.556, 51.153]
  Set speed (120.0 mm/s)
  MoveL 8857 to (502.59, 503.19, 17.4) mm, rotated rx 0 ry 90 rz 0 deg; joints [-12.249, -28.064, 111.255, -16.286, -82.6, 51.133]
  Set speed (15.0 mm/s)
  Call Extruder(0.050)
  MoveL 8858 to (501.37, 504.42, 17.4) mm, rotated rx 0 ry 90 rz 0 deg; joints [-12.385, -28.082, 111.37, -16.419, -82.697, 51.122]
  Set speed (120.0 mm/s)
  MoveL 8859 to (501.03, 504.76, 17.4) mm, rotated rx 0 ry 90 rz 0 deg; joints [-12.423, -28.087, 111.401, -16.456, -82.723, 51.118]
  Set speed (15.0 mm/s)
  Call Extruder(0.066)
  MoveL 8860 to (499.43, 506.36, 17.4) mm, rotated rx 0 ry 90 rz 0 deg; joints [-12.602, -28.111, 111.55, -16.632, -82.849, 51.102]
  Set speed (120.0 mm/s)
  MoveL 8861 to (498.44, 506.36, 17.4) mm, rotated rx 0 ry 90 rz 0 deg; joints [-12.622, -28.13, 111.668, -16.649, -82.945, 51.076]
  Set speed (15.0 mm/s)
  MoveL 8862 to (500.04, 504.76, 17.4) mm, rotated rx 0 ry 90 rz 0 deg; joints [-12.443, -28.106, 111.52, -16.473, -82.819, 51.092]
  Set speed (120.0 mm/s)
  MoveL 8863 to (499.05, 504.76, 17.4) mm, rotated rx 0 ry 90 rz 0 deg; joints [-12.463, -28.125, 111.638, -16.489, -82.915, 51.066]
  Set speed (15.0 mm/s)
  MoveL 8864 to (497.45, 506.36, 17.4) mm, rotated rx 0 ry 90 rz 0 deg; joints [-12.642, -28.148, 111.786, -16.666, -83.041, 51.049]
  Set speed (120.0 mm/s)
  MoveL 8865 to (496.46, 506.36, 17.4) mm, rotated rx 0 ry 90 rz 0 deg; joints [-12.663, -28.167, 111.904, -16.683, -83.136, 51.023]
  Set speed (15.0 mm/s)
  MoveL 8866 to (498.06, 504.76, 17.4) mm, rotated rx 0 ry 90 rz 0 deg; joints [-12.483, -28.144, 111.756, -16.506, -83.011, 51.04]
  Set speed (120.0 mm/s)
  MoveL 8867 to (497.07, 504.76, 17.4) mm, rotated rx 0 ry 90 rz 0 deg; joints [-12.503, -28.162, 111.874, -16.523, -83.107, 51.013]
  Set speed (15.0 mm/s)
  Call Extruder(0.029)
  MoveL 8868 to (496.36, 505.47, 17.4) mm, rotated rx 0 ry 90 rz 0 deg; joints [-12.583, -28.172, 111.939, -16.601, -83.162, 51.006]
  Set speed (120.0 mm/s)
  MoveL 8869 to (500.7, 503.11, 17.4) mm, rotated rx 0 ry 90 rz 0 deg; joints [-12.279, -28.1, 111.484, -16.309, -82.785, 51.082]
  Set speed (15.0 mm/s)
  Call Extruder(0.050)
  MoveL 8870 to (501.92, 501.88, 17.4) mm, rotated rx 0 ry 90 rz 0 deg; joints [-12.143, -28.082, 111.369, -16.175, -82.688, 51.094]
  Set speed (120.0 mm/s)
  MoveL 8871 to (501.59, 501.23, 17.4) mm, rotated rx 0 ry 90 rz 0 deg; joints [-12.09, -28.091, 111.426, -16.12, -82.732, 51.075]
  Set speed (15.0 mm/s)
  MoveL 8872 to (500.36, 502.45, 17.4) mm, rotated rx 0 ry 90 rz 0 deg; joints [-12.226, -28.11, 111.541, -16.254, -82.829, 51.063]
  Set speed (120.0 mm/s)
  MoveL 8873 to (500.03, 501.8, 17.4) mm, rotated rx 0 ry 90 rz 0 deg; joints [-12.172, -28.119, 111.598, -16.198, -82.873, 51.044]
  Set speed (15.0 mm/s)
  Call Extruder(0.050)
  MoveL 8874 to (501.25, 500.58, 17.4) mm, rotated rx 0 ry 90 rz 0 deg; joints [-12.037, -28.1, 111.483, -16.065, -82.777, 51.056]
  Set speed (120.0 mm/s)
  MoveL 8875 to (500.92, 499.92, 17.4) mm, rotated rx 0 ry 90 rz 0 deg; joints [-11.983, -28.109, 111.54, -16.009, -82.821, 51.036]
  Set speed (15.0 mm/s)
  Call Extruder(0.050)
